C07285=1085.973,384.682,401.818,177.153,26.555,154.362
C07286=1085.978,384.905,401.783,177.157,26.561,154.363
C07287=1085.983,385.128,401.749,177.160,26.567,154.364
C07288=1085.989,385.351,401.714,177.163,26.574,154.365
C07289=1085.995,385.598,401.676,177.166,26.581,154.367
C07290=1086.002,385.844,401.637,177.169,26.588,154.368
C07291=1086.008,386.091,401.600,177.172,26.595,154.369
C07292=1086.014,386.339,401.561,177.176,26.602,154.371
C07293=1086.020,386.585,401.523,177.179,26.608,154.372
C07294=1086.027,386.832,401.485,177.183,26.615,154.373
C07295=1086.032,387.079,401.447,177.186,26.622,154.374
C07296=1086.039,387.326,401.408,177.189,26.629,154.376
C07297=1086.045,387.573,401.370,177.193,26.637,154.377
C07298=1086.052,387.820,401.331,177.196,26.644,154.378
C07299=1086.057,388.066,401.293,177.200,26.651,154.380
C07300=1086.064,388.314,401.254,177.203,26.658,154.381
C07301=1086.069,388.560,401.216,177.206,26.665,154.383
C07302=1086.076,388.807,401.177,177.210,26.672,154.384
C07303=1086.082,389.054,401.140,177.213,26.680,154.385
C07304=1086.089,389.301,401.101,177.217,26.687,154.387
C07305=1086.095,389.548,401.061,177.220,26.694,154.388
C07306=1086.101,389.795,401.024,177.223,26.701,154.389
C07307=1086.108,390.041,400.985,177.227,26.709,154.391
C07308=1086.115,390.288,400.946,177.230,26.715,154.392
C07309=1086.120,390.535,400.908,177.233,26.723,154.393
C07310=1086.127,390.782,400.869,177.237,26.730,154.395
C07311=1086.133,391.028,400.830,177.240,26.737,154.396
C07312=1086.139,391.276,400.792,177.244,26.745,154.398
C07313=1086.145,391.523,400.753,177.247,26.752,154.399
C07314=1086.152,391.769,400.714,177.250,26.759,154.400
C07315=1086.158,392.016,400.675,177.254,26.767,154.402
C07316=1086.164,392.263,400.636,177.257,26.774,154.403
C07317=1086.171,392.509,400.597,177.260,26.781,154.405
C07318=1086.176,392.757,400.559,177.264,26.789,154.406
C07319=1086.183,393.004,400.520,177.267,26.796,154.408
C07320=1086.189,393.251,400.480,177.270,26.804,154.409
C07321=1086.196,393.497,400.442,177.274,26.812,154.411
C07322=1086.202,393.744,400.403,177.277,26.819,154.412
C07323=1086.208,393.991,400.364,177.280,26.826,154.413
C07324=1086.214,394.237,400.325,177.284,26.834,154.415
C07325=1086.221,394.484,400.286,177.287,26.842,154.416
C07326=1086.227,394.731,400.246,177.290,26.849,154.418
C07327=1086.234,394.978,400.208,177.294,26.857,154.419
C07328=1086.240,395.225,400.168,177.298,26.865,154.421
C07329=1086.246,395.471,400.129,177.301,26.873,154.422
C07330=1086.252,395.718,400.090,177.305,26.880,154.424
C07331=1086.258,395.965,400.050,177.308,26.888,154.425
C07332=1086.265,396.212,400.011,177.311,26.895,154.427
C07333=1086.271,396.459,399.972,177.315,26.903,154.428
C07334=1086.277,396.705,399.933,177.318,26.911,154.430
C07335=1086.284,396.951,399.893,177.321,26.919,154.431
C07336=1086.290,397.199,399.854,177.325,26.927,154.433
C07337=1086.296,397.429,399.817,177.328,26.934,154.434
C07338=1086.302,397.658,399.780,177.331,26.941,154.436
C07339=1086.307,397.887,399.744,177.335,26.949,154.437
C07340=1086.314,398.117,399.707,177.337,26.956,154.439
C07341=1086.319,398.347,399.670,177.340,26.964,154.440
C07342=1086.325,398.577,399.633,177.344,26.971,154.442
C07343=1086.331,398.806,399.597,177.347,26.978,154.443
C07344=1086.337,399.036,399.560,177.351,26.986,154.444
C07345=1086.343,399.283,399.520,177.354,26.994,154.446
C07346=1086.350,399.530,399.480,177.357,27.002,154.448
C07347=1086.356,399.777,399.441,177.360,27.010,154.449
C07348=1086.362,400.023,399.401,177.364,27.018,154.451
C07349=1086.368,400.270,399.361,177.367,27.026,154.453
C07350=1086.375,400.517,399.322,177.371,27.034,154.454
C07351=1086.381,400.764,399.282,177.374,27.043,154.456
C07352=1086.388,401.010,399.242,177.378,27.050,154.457
C07353=1086.394,401.257,399.202,177.381,27.059,154.459
C07354=1086.400,401.504,399.162,177.384,27.067,154.461
C07355=1086.407,401.750,399.122,177.388,27.075,154.462
C07356=1086.413,401.997,399.082,177.392,27.084,154.464
C07357=1086.419,402.244,399.043,177.395,27.092,154.466
C07358=1086.425,402.491,399.003,177.398,27.100,154.467
C07359=1086.432,402.737,398.962,177.402,27.108,154.469
C07360=1086.438,402.984,398.922,177.406,27.117,154.471
C07361=1086.445,403.230,398.882,177.409,27.125,154.472
C07362=1086.451,403.477,398.843,177.412,27.133,154.474
C07363=1086.457,403.724,398.803,177.416,27.142,154.476
C07364=1086.463,403.970,398.762,177.420,27.150,154.477
C07365=1086.470,404.217,398.722,177.423,27.159,154.479
C07366=1086.477,404.464,398.682,177.427,27.168,154.481
C07367=1086.483,404.711,398.642,177.430,27.176,154.482
C07368=1086.490,404.957,398.601,177.433,27.184,154.484
C07369=1086.496,405.204,398.561,177.437,27.193,154.486
C07370=1086.502,405.450,398.521,177.441,27.202,154.488
C07371=1086.509,405.697,398.481,177.444,27.211,154.489
C07372=1086.515,405.944,398.440,177.447,27.219,154.491
C07373=1086.521,406.191,398.400,177.451,27.228,154.493
C07374=1086.528,406.437,398.360,177.455,27.236,154.495
C07375=1086.534,406.684,398.319,177.459,27.245,154.496
C07376=1086.540,406.930,398.279,177.462,27.254,154.498
C07377=1086.547,407.177,398.237,177.465,27.263,154.500
C07378=1086.553,407.424,398.197,177.469,27.272,154.502
C07379=1086.560,407.670,398.157,177.472,27.281,154.504
C07380=1086.566,407.917,398.117,177.476,27.290,154.505
C07381=1086.573,408.164,398.075,177.480,27.299,154.507
C07382=1086.579,408.410,398.035,177.483,27.307,154.509
C07383=1086.585,408.657,397.994,177.487,27.316,154.511
C07384=1086.591,408.903,397.953,177.490,27.325,154.513
C07385=1086.598,409.150,397.913,177.494,27.335,154.515
C07386=1086.604,409.397,397.872,177.497,27.343,154.516
C07387=1086.611,409.643,397.831,177.501,27.352,154.518
C07388=1086.616,409.890,397.791,177.505,27.362,154.520
C07389=1086.624,410.136,397.749,177.508,27.371,154.522
C07390=1086.630,410.383,397.709,177.512,27.380,154.524
C07391=1086.636,410.629,397.668,177.515,27.389,154.526
C07392=1086.643,410.876,397.627,177.519,27.398,154.528
C07393=1086.649,411.106,397.589,177.523,27.407,154.529
C07394=1086.655,411.336,397.550,177.526,27.415,154.531
C07395=1086.661,411.567,397.512,177.529,27.424,154.533
C07396=1086.667,411.797,397.474,177.532,27.433,154.535
C07397=1086.673,412.028,397.435,177.536,27.442,154.537
C07398=1086.679,412.258,397.396,177.540,27.451,154.538
C07399=1086.685,412.489,397.359,177.543,27.459,154.540
C07400=1086.691,412.719,397.320,177.546,27.468,154.542
C07401=1086.698,412.966,397.279,177.550,27.478,154.544
C07402=1086.704,413.212,397.238,177.553,27.487,154.546
C07403=1086.712,413.458,397.196,177.558,27.496,154.548
C07404=1086.717,413.705,397.155,177.561,27.505,154.550
C07405=1086.724,413.952,397.114,177.565,27.515,154.552
C07406=1086.730,414.198,397.073,177.568,27.525,154.554
C07407=1086.738,414.445,397.032,177.572,27.534,154.556
C07408=1086.744,414.691,396.990,177.576,27.544,154.558
C07409=1086.751,414.937,396.949,177.579,27.553,154.560
C07410=1086.757,415.184,396.908,177.583,27.563,154.562
C07411=1086.763,415.431,396.866,177.587,27.573,154.564
C07412=1086.770,415.676,396.825,177.590,27.582,154.566
C07413=1086.777,415.923,396.783,177.595,27.592,154.568
C07414=1086.784,416.170,396.742,177.599,27.602,154.570
C07415=1086.790,416.416,396.700,177.602,27.612,154.572
C07416=1086.797,416.662,396.658,177.606,27.622,154.574
C07417=1086.803,416.909,396.616,177.610,27.632,154.576
C07418=1086.809,417.156,396.574,177.613,27.641,154.578
C07419=1086.816,417.401,396.534,177.617,27.652,154.580
C07420=1086.823,417.648,396.491,177.621,27.662,154.582
C07421=1086.829,417.895,396.449,177.624,27.671,154.584
C07422=1086.835,418.141,396.408,177.628,27.682,154.587
C07423=1086.842,418.388,396.366,177.632,27.692,154.589
C07424=1086.848,418.633,396.324,177.636,27.702,154.591
C07425=1086.855,418.880,396.283,177.639,27.712,154.593
C07426=1086.862,419.126,396.240,177.643,27.722,154.595
C07427=1086.868,419.372,396.199,177.647,27.733,154.597
C07428=1086.875,419.619,396.156,177.651,27.743,154.599
C07429=1086.882,419.866,396.114,177.654,27.753,154.602
C07430=1086.888,420.112,396.072,177.658,27.764,154.604
C07431=1086.894,420.358,396.030,177.662,27.774,154.606
C07432=1086.901,420.604,395.988,177.666,27.784,154.608
C07433=1086.909,420.851,395.946,177.670,27.795,154.610
C07434=1086.915,421.097,395.904,177.673,27.805,154.613
C07435=1086.922,421.343,395.862,177.677,27.815,154.615
C07436=1086.928,421.590,395.820,177.681,27.826,154.617
C07437=1086.935,421.836,395.777,177.685,27.836,154.619
C07438=1086.942,422.082,395.735,177.689,27.847,154.622
C07439=1086.949,422.329,395.692,177.693,27.858,154.624
C07440=1086.955,422.575,395.651,177.697,27.868,154.626
C07441=1086.962,422.821,395.608,177.700,27.879,154.628
C07442=1086.968,423.067,395.566,177.704,27.890,154.631
C07443=1086.975,423.314,395.523,177.708,27.901,154.633
C07444=1086.981,423.560,395.480,177.712,27.912,154.635
C07445=1086.988,423.806,395.438,177.716,27.922,154.638
C07446=1086.995,424.052,395.395,177.720,27.933,154.640
C07447=1087.001,424.298,395.353,177.724,27.944,154.642
C07448=1087.008,424.545,395.310,177.728,27.955,154.645
C07449=1087.015,424.783,395.269,177.732,27.966,154.647
C07450=1087.021,425.021,395.228,177.735,27.976,154.649
C07451=1087.028,425.260,395.186,177.739,27.987,154.651
C07452=1087.034,425.497,395.145,177.743,27.998,154.654
C07453=1087.041,425.736,395.104,177.748,28.009,154.656
C07454=1087.047,425.973,395.062,177.751,28.019,154.658
C07455=1087.054,426.212,395.021,177.755,28.030,154.661
C07456=1087.060,426.451,394.979,177.759,28.041,154.663
C07457=1087.067,426.697,394.936,177.763,28.052,154.665
C07458=1087.074,426.943,394.893,177.767,28.063,154.668
C07459=1087.081,427.189,394.850,177.771,28.074,154.670
C07460=1087.087,427.435,394.807,177.774,28.086,154.673
C07461=1087.094,427.681,394.764,177.778,28.097,154.675
C07462=1087.101,427.927,394.721,177.782,28.108,154.678
C07463=1087.108,428.173,394.678,177.786,28.120,154.680
C07464=1087.114,428.420,394.635,177.790,28.131,154.683
C07465=1087.121,428.665,394.592,177.795,28.143,154.685
C07466=1087.128,428.912,394.549,177.799,28.154,154.688
C07467=1087.134,429.158,394.505,177.803,28.166,154.690
C07468=1087.141,429.404,394.463,177.807,28.178,154.693
C07469=1087.148,429.650,394.419,177.811,28.190,154.695
C07470=1087.155,429.896,394.376,177.815,28.201,154.698
C07471=1087.161,430.141,394.332,177.819,28.213,154.700
C07472=1087.168,430.388,394.289,177.823,28.225,154.703
C07473=1087.175,430.634,394.246,177.827,28.236,154.706
C07474=1087.182,430.880,394.202,177.832,28.249,154.708
C07475=1087.189,431.126,394.158,177.836,28.261,154.711
C07476=1087.196,431.372,394.116,177.839,28.273,154.714
C07477=1087.202,431.618,394.072,177.843,28.284,154.716
C07478=1087.209,431.864,394.028,177.847,28.297,154.719
C07479=1087.216,432.110,393.985,177.852,28.309,154.721
C07480=1087.223,432.357,393.940,177.856,28.321,154.724
C07481=1087.230,432.602,393.897,177.860,28.333,154.727
C07482=1087.236,432.848,393.853,177.864,28.345,154.729
C07483=1087.243,433.094,393.810,177.869,28.357,154.732
C07484=1087.250,433.341,393.766,177.873,28.370,154.735
C07485=1087.257,433.586,393.721,177.877,28.382,154.738
C07486=1087.264,433.832,393.677,177.881,28.394,154.740
C07487=1087.271,434.078,393.634,177.885,28.407,154.743
C07488=1087.278,434.324,393.590,177.889,28.420,154.746
C07489=1087.284,434.570,393.546,177.893,28.432,154.749
C07490=1087.291,434.816,393.502,177.897,28.444,154.751
C07491=1087.297,435.062,393.458,177.902,28.457,154.754
C07492=1087.305,435.308,393.414,177.906,28.470,154.757
C07493=1087.312,435.553,393.369,177.910,28.483,154.760
C07494=1087.318,435.799,393.326,177.915,28.495,154.763
C07495=1087.326,436.045,393.281,177.919,28.508,154.765
C07496=1087.332,436.291,393.237,177.922,28.521,154.768
C07497=1087.339,436.537,393.192,177.927,28.534,154.771
C07498=1087.346,436.783,393.149,177.931,28.547,154.774
C07499=1087.353,437.028,393.104,177.936,28.560,154.777
C07500=1087.360,437.275,393.060,177.940,28.573,154.780
C07501=1087.367,437.520,393.015,177.944,28.586,154.783
C07502=1087.374,437.766,392.970,177.949,28.599,154.786
C07503=1087.381,438.012,392.926,177.952,28.612,154.789
C07504=1087.388,438.258,392.882,177.957,28.625,154.792
C07505=1087.395,438.502,392.837,177.961,28.638,154.795
C07506=1087.402,438.746,392.793,177.966,28.652,154.797
C07507=1087.409,438.990,392.749,177.970,28.665,154.800
C07508=1087.416,439.234,392.704,177.974,28.678,154.803
C07509=1087.423,439.478,392.660,177.979,28.691,154.806
C07510=1087.430,439.723,392.616,177.983,28.704,154.809
C07511=1087.438,439.967,392.572,177.988,28.718,154.812
C07512=1087.444,440.211,392.527,177.991,28.731,154.815
C07513=1087.451,440.457,392.482,177.996,28.745,154.818
C07514=1087.458,440.702,392.437,178.000,28.758,154.822
C07515=1087.465,440.948,392.393,178.005,28.772,154.825
C07516=1087.473,441.194,392.348,178.009,28.786,154.828
C07517=1087.479,441.440,392.302,178.014,28.800,154.831
C07518=1087.486,441.685,392.257,178.019,28.814,154.834
C07519=1087.493,441.931,392.212,178.022,28.828,154.837
C07520=1087.500,442.177,392.167,178.027,28.842,154.840
C07521=1087.508,442.422,392.122,178.031,28.855,154.843
C07522=1087.515,442.667,392.077,178.036,28.869,154.847
C07523=1087.521,442.914,392.032,178.041,28.884,154.850
C07524=1087.529,443.159,391.986,178.045,28.898,154.853
C07525=1087.536,443.405,391.941,178.050,28.912,154.856
C07526=1087.543,443.650,391.895,178.054,28.927,154.860
C07527=1087.550,443.896,391.850,178.058,28.941,154.863
C07528=1087.558,444.142,391.805,178.063,28.955,154.866
C07529=1087.564,444.387,391.760,178.068,28.970,154.869
C07530=1087.571,444.633,391.714,178.072,28.984,154.873
C07531=1087.579,444.878,391.668,178.077,28.999,154.876
C07532=1087.586,445.124,391.623,178.081,29.013,154.879
C07533=1087.593,445.370,391.577,178.085,29.028,154.883
C07534=1087.601,445.616,391.531,178.089,29.042,154.886
C07535=1087.607,445.861,391.486,178.092,29.057,154.890
C07536=1087.614,446.107,391.440,178.096,29.071,154.893
C07537=1087.621,446.352,391.394,178.099,29.085,154.896
C07538=1087.629,446.598,391.349,178.102,29.100,154.900
C07539=1087.636,446.844,391.302,178.105,29.114,154.903
C07540=1087.643,447.089,391.257,178.108,29.129,154.907
C07541=1087.650,447.335,391.210,178.111,29.143,154.910
C07542=1087.658,447.580,391.165,178.113,29.158,154.914
C07543=1087.665,447.826,391.119,178.115,29.172,154.917
C07544=1087.673,448.071,391.073,178.117,29.187,154.921
C07545=1087.679,448.317,391.027,178.119,29.201,154.924
C07546=1087.687,448.563,390.981,178.120,29.215,154.928
C07547=1087.694,448.808,390.935,178.122,29.229,154.931
C07548=1087.701,449.054,390.888,178.123,29.244,154.935
C07549=1087.708,449.299,390.843,178.124,29.258,154.938
C07550=1087.716,449.544,390.797,178.125,29.272,154.942
C07551=1087.724,449.789,390.751,178.126,29.286,154.945
C07552=1087.735,450.036,390.706,178.127,29.299,154.948
C07553=1087.357,450.027,390.509,178.088,29.488,155.000
C07554=1087.346,449.781,390.554,178.087,29.475,154.997
C07555=1087.338,449.535,390.600,178.086,29.461,154.993
C07556=1087.330,449.290,390.646,178.085,29.447,154.990
C07557=1087.323,449.046,390.691,178.084,29.433,154.986
C07558=1087.314,448.745,390.748,178.082,29.416,154.982
C07559=1087.305,448.446,390.804,178.080,29.398,154.978
C07560=1087.296,448.146,390.861,178.077,29.380,154.973
C07561=1087.287,447.846,390.917,178.076,29.363,154.969
C07562=1087.280,447.601,390.963,178.073,29.348,154.965
C07563=1087.273,447.355,391.009,178.071,29.334,154.962
C07564=1087.265,447.110,391.055,178.069,29.320,154.958
C07565=1087.258,446.864,391.101,178.066,29.305,154.955
C07566=1087.251,446.618,391.147,178.062,29.291,154.952
C07567=1087.244,446.373,391.193,178.059,29.276,154.948
C07568=1087.236,446.127,391.239,178.055,29.261,154.945
C07569=1087.230,445.882,391.285,178.052,29.247,154.941
C07570=1087.222,445.637,391.330,178.048,29.233,154.938
C07571=1087.215,445.391,391.377,178.045,29.218,154.934
C07572=1087.208,445.145,391.421,178.040,29.203,154.931
C07573=1087.200,444.899,391.467,178.036,29.188,154.928
C07574=1087.194,444.654,391.513,178.032,29.174,154.924
C07575=1087.186,444.408,391.558,178.027,29.160,154.921
C07576=1087.179,444.162,391.604,178.022,29.145,154.918
C07577=1087.172,443.917,391.650,178.018,29.131,154.914
C07578=1087.165,443.671,391.695,178.013,29.117,154.911
C07579=1087.157,443.426,391.740,178.008,29.102,154.908
C07580=1087.150,443.180,391.787,178.004,29.088,154.905
C07581=1087.144,442.935,391.831,177.999,29.074,154.901
C07582=1087.136,442.689,391.876,177.994,29.059,154.898
C07583=1087.129,442.443,391.922,177.990,29.045,154.895
C07584=1087.123,442.197,391.967,177.985,29.031,154.892
C07585=1087.115,441.952,392.013,177.981,29.017,154.889
C07586=1087.108,441.706,392.058,177.976,29.003,154.885
C07587=1087.100,441.460,392.102,177.972,28.990,154.882
C07588=1087.093,441.215,392.148,177.967,28.976,154.879
C07589=1087.086,440.969,392.193,177.962,28.962,154.876
C07590=1087.080,440.724,392.238,177.958,28.948,154.873
C07591=1087.073,440.477,392.283,177.953,28.934,154.870
C07592=1087.065,440.231,392.328,177.949,28.921,154.867
C07593=1087.059,439.986,392.372,177.945,28.907,154.864
C07594=1087.053,439.776,392.411,177.941,28.896,154.861
C07595=1087.046,439.566,392.449,177.937,28.884,154.858
C07596=1087.040,439.356,392.488,177.934,28.873,154.856
C07597=1087.034,439.146,392.525,177.929,28.861,154.853
C07598=1087.028,438.936,392.563,177.926,28.850,154.851
C07599=1087.022,438.725,392.603,177.922,28.839,154.848
C07600=1087.016,438.515,392.640,177.919,28.827,154.846
C07601=1087.010,438.305,392.678,177.914,28.816,154.843
C07602=1087.003,438.059,392.723,177.910,28.803,154.840
C07603=1086.995,437.814,392.767,177.905,28.789,154.837
C07604=1086.988,437.568,392.812,177.902,28.776,154.834
C07605=1086.981,437.322,392.856,177.897,28.763,154.831
C07606=1086.975,437.076,392.901,177.893,28.750,154.828
C07607=1086.967,436.830,392.946,177.889,28.737,154.826
C07608=1086.961,436.584,392.989,177.884,28.724,154.823
C07609=1086.954,436.339,393.034,177.880,28.711,154.820
C07610=1086.947,436.093,393.079,177.876,28.699,154.817
C07611=1086.940,435.847,393.122,177.871,28.685,154.814
C07612=1086.932,435.601,393.167,177.867,28.673,154.811
C07613=1086.926,435.355,393.211,177.863,28.660,154.808
C07614=1086.920,435.109,393.255,177.858,28.647,154.806
C07615=1086.912,434.863,393.300,177.854,28.635,154.803
C07616=1086.905,434.618,393.343,177.850,28.622,154.800
C07617=1086.898,434.372,393.388,177.845,28.609,154.797
C07618=1086.891,434.126,393.432,177.841,28.597,154.794
C07619=1086.885,433.880,393.476,177.837,28.585,154.792
C07620=1086.878,433.634,393.519,177.833,28.572,154.789
C07621=1086.871,433.389,393.563,177.828,28.560,154.786
C07622=1086.864,433.142,393.608,177.824,28.547,154.783
C07623=1086.858,432.896,393.651,177.820,28.535,154.781
C07624=1086.851,432.650,393.695,177.816,28.523,154.778
C07625=1086.843,432.404,393.739,177.811,28.510,154.775
C07626=1086.837,432.158,393.783,177.807,28.498,154.773
C07627=1086.830,431.912,393.826,177.803,28.486,154.770
C07628=1086.823,431.666,393.870,177.799,28.474,154.767
C07629=1086.816,431.420,393.913,177.795,28.462,154.765
C07630=1086.809,431.174,393.957,177.790,28.450,154.762
C07631=1086.802,430.928,394.001,177.786,28.438,154.760
C07632=1086.796,430.682,394.044,177.782,28.426,154.757
C07633=1086.788,430.436,394.088,177.778,28.414,154.754
C07634=1086.782,430.190,394.131,177.774,28.403,154.752
C07635=1086.775,429.944,394.174,177.770,28.391,154.749
C07636=1086.768,429.697,394.218,177.766,28.379,154.746
C07637=1086.761,429.452,394.262,177.761,28.367,154.744
C07638=1086.755,429.205,394.305,177.757,28.355,154.741
C07639=1086.748,428.959,394.348,177.753,28.343,154.739
C07640=1086.741,428.713,394.392,177.749,28.332,154.736
C07641=1086.734,428.467,394.434,177.745,28.321,154.734
C07642=1086.728,428.221,394.478,177.741,28.309,154.731
C07643=1086.721,427.975,394.521,177.737,28.298,154.729
C07644=1086.714,427.729,394.564,177.733,28.286,154.726
C07645=1086.707,427.483,394.607,177.729,28.275,154.724
C07646=1086.701,427.237,394.650,177.725,28.263,154.721
C07647=1086.694,426.991,394.693,177.721,28.252,154.719
C07648=1086.687,426.745,394.736,177.717,28.241,154.717
C07649=1086.680,426.499,394.779,177.713,28.230,154.714
C07650=1086.673,426.259,394.821,177.709,28.218,154.712
C07651=1086.666,426.021,394.863,177.705,28.208,154.709
C07652=1086.660,425.782,394.904,177.700,28.197,154.707
C07653=1086.654,425.543,394.946,177.697,28.186,154.705
C07654=1086.647,425.305,394.987,177.693,28.175,154.702
C07655=1086.641,425.065,395.028,177.689,28.165,154.700
C07656=1086.634,424.827,395.069,177.685,28.154,154.698
C07657=1086.628,424.588,395.112,177.682,28.143,154.695
C07658=1086.621,424.342,395.154,177.678,28.133,154.693
C07659=1086.614,424.095,395.197,177.674,28.121,154.691
C07660=1086.607,423.849,395.239,177.670,28.110,154.688
C07661=1086.601,423.603,395.282,177.666,28.100,154.686
C07662=1086.594,423.357,395.324,177.662,28.089,154.684
C07663=1086.588,423.111,395.367,177.658,28.078,154.682
C07664=1086.581,422.864,395.410,177.654,28.067,154.679
C07665=1086.575,422.618,395.452,177.649,28.056,154.677
C07666=1086.568,422.372,395.495,177.646,28.046,154.675
C07667=1086.561,422.126,395.537,177.642,28.035,154.672
C07668=1086.555,421.880,395.579,177.638,28.025,154.670
C07669=1086.548,421.633,395.621,177.634,28.014,154.668
C07670=1086.541,421.387,395.664,177.630,28.003,154.666
C07671=1086.534,421.141,395.706,177.626,27.993,154.663
C07672=1086.527,420.894,395.749,177.623,27.983,154.661
C07673=1086.521,420.647,395.791,177.619,27.972,154.659
C07674=1086.515,420.402,395.833,177.615,27.962,154.657
C07675=1086.508,420.155,395.875,177.611,27.951,154.654
C07676=1086.500,419.909,395.917,177.607,27.941,154.652
C07677=1086.494,419.663,395.959,177.603,27.931,154.650
C07678=1086.488,419.416,396.001,177.599,27.920,154.648
C07679=1086.481,419.170,396.043,177.595,27.910,154.646
C07680=1086.474,418.923,396.085,177.591,27.900,154.644
C07681=1086.468,418.678,396.127,177.588,27.890,154.641
C07682=1086.461,418.431,396.169,177.584,27.879,154.639
C07683=1086.454,418.185,396.211,177.580,27.869,154.637
C07684=1086.448,417.939,396.252,177.576,27.859,154.635
C07685=1086.441,417.692,396.294,177.573,27.849,154.633
C07686=1086.435,417.445,396.337,177.569,27.839,154.631
C07687=1086.429,417.199,396.378,177.564,27.829,154.629
C07688=1086.422,416.952,396.420,177.561,27.819,154.627
C07689=1086.415,416.706,396.461,177.557,27.809,154.625
C07690=1086.408,416.460,396.503,177.553,27.799,154.622
C07691=1086.402,416.213,396.545,177.550,27.789,154.620
C07692=1086.396,415.967,396.587,177.546,27.780,154.618
C07693=1086.389,415.720,396.628,177.542,27.770,154.616
C07694=1086.383,415.474,396.669,177.538,27.760,154.614
C07695=1086.376,415.227,396.711,177.534,27.750,154.612
C07696=1086.369,414.981,396.752,177.531,27.741,154.610
C07697=1086.363,414.734,396.794,177.527,27.731,154.608
C07698=1086.356,414.488,396.835,177.523,27.721,154.606
C07699=1086.350,414.242,396.876,177.520,27.712,154.604
C07700=1086.342,413.995,396.918,177.516,27.702,154.602
C07701=1086.336,413.749,396.959,177.512,27.693,154.600
C07702=1086.329,413.502,397.000,177.508,27.683,154.598
C07703=1086.323,413.256,397.042,177.504,27.673,154.596
C07704=1086.316,413.009,397.083,177.501,27.664,154.594
C07705=1086.310,412.763,397.125,177.497,27.654,154.592
C07706=1086.303,412.531,397.163,177.493,27.646,154.591
C07707=1086.297,412.301,397.201,177.490,27.637,154.589
C07708=1086.292,412.070,397.240,177.487,27.628,154.587
C07709=1086.285,411.839,397.279,177.483,27.620,154.585
C07710=1086.279,411.608,397.316,177.479,27.611,154.583
C07711=1086.273,411.377,397.356,177.476,27.602,154.582
C07712=1086.267,411.146,397.394,177.473,27.593,154.580
C07713=1086.260,410.915,397.433,177.469,27.584,154.578
C07714=1086.255,410.668,397.473,177.466,27.575,154.576
C07715=1086.248,410.423,397.514,177.462,27.566,154.574
C07716=1086.242,410.175,397.555,177.459,27.557,154.572
C07717=1086.235,409.929,397.596,177.455,27.548,154.570
C07718=1086.229,409.683,397.636,177.451,27.539,154.568
C07719=1086.222,409.436,397.678,177.447,27.530,154.567
C07720=1086.216,409.189,397.718,177.444,27.520,154.565
C07721=1086.210,408.943,397.760,177.440,27.511,154.563
C07722=1086.203,408.696,397.800,177.437,27.502,154.561
C07723=1086.196,408.450,397.841,177.433,27.493,154.559
C07724=1086.191,408.203,397.882,177.429,27.484,154.557
C07725=1086.184,407.956,397.922,177.426,27.476,154.556
C07726=1086.178,407.710,397.964,177.423,27.466,154.554
C07727=1086.171,407.463,398.004,177.419,27.457,154.552
C07728=1086.165,407.217,398.044,177.415,27.449,154.550
C07729=1086.158,406.970,398.084,177.411,27.440,154.548
C07730=1086.152,406.723,398.126,177.408,27.431,154.547
C07731=1086.146,406.477,398.166,177.405,27.422,154.545
C07732=1086.139,406.230,398.206,177.400,27.413,154.543
C07733=1086.133,405.984,398.246,177.397,27.405,154.541
C07734=1086.126,405.737,398.287,177.394,27.396,154.539
C07735=1086.120,405.490,398.328,177.390,27.387,154.538
C07736=1086.114,405.243,398.368,177.386,27.379,154.536
C07737=1086.107,404.997,398.408,177.383,27.370,154.534
C07738=1086.101,404.750,398.448,177.379,27.362,154.533
C07739=1086.095,404.503,398.488,177.376,27.353,154.531
C07740=1086.088,404.256,398.529,177.372,27.345,154.529
C07741=1086.081,404.010,398.569,177.369,27.336,154.527
C07742=1086.075,403.763,398.609,177.365,27.327,154.526
C07743=1086.069,403.517,398.649,177.362,27.319,154.524
C07744=1086.062,403.270,398.689,177.358,27.311,154.522
C07745=1086.056,403.024,398.730,177.355,27.302,154.520
C07746=1086.049,402.777,398.770,177.351,27.294,154.519
C07747=1086.043,402.530,398.809,177.347,27.285,154.517
C07748=1086.036,402.283,398.850,177.344,27.277,154.515
C07749=1086.030,402.036,398.890,177.341,27.269,154.514
C07750=1086.024,401.790,398.930,177.337,27.261,154.512
C07751=1086.017,401.543,398.970,177.333,27.252,154.511
C07752=1086.011,401.296,399.010,177.330,27.244,154.509
C07753=1086.005,401.050,399.050,177.327,27.236,154.507
C07754=1085.998,400.803,399.090,177.323,27.228,154.506
C07755=1085.992,400.556,399.129,177.319,27.219,154.504
C07756=1085.985,400.310,399.169,177.316,27.211,154.502
C07757=1085.979,400.063,399.208,177.313,27.203,154.501
C07758=1085.973,399.816,399.248,177.309,27.195,154.499
C07759=1085.967,399.569,399.288,177.306,27.187,154.497
C07760=1085.960,399.322,399.328,177.303,27.179,154.496
C07761=1085.954,399.075,399.367,177.298,27.170,154.494
C07762=1085.948,398.845,399.404,177.296,27.163,154.493
C07763=1085.942,398.615,399.441,177.292,27.156,154.491
C07764=1085.936,398.385,399.479,177.289,27.148,154.490
C07765=1085.931,398.156,399.515,177.286,27.141,154.488
C07766=1085.925,397.925,399.552,177.283,27.134,154.487
C07767=1085.918,397.695,399.589,177.280,27.126,154.486
C07768=1085.913,397.465,399.626,177.276,27.119,154.484
C07769=1085.907,397.235,399.663,177.273,27.111,154.483
C07770=1085.900,396.988,399.702,177.269,27.103,154.481
C07771=1085.894,396.741,399.741,177.266,27.096,154.480
C07772=1085.888,396.493,399.781,177.263,27.088,154.478
C07773=1085.882,396.248,399.821,177.259,27.080,154.476
C07774=1085.875,396.001,399.859,177.256,27.072,154.475
C07775=1085.869,395.754,399.899,177.253,27.065,154.473
C07776=1085.863,395.507,399.938,177.249,27.057,154.472
C07777=1085.856,395.260,399.977,177.246,27.049,154.470
C07778=1085.850,395.014,400.017,177.242,27.041,154.469
C07779=1085.844,394.767,400.056,177.238,27.033,154.467
C07780=1085.838,394.520,400.095,177.235,27.026,154.466
C07781=1085.831,394.273,400.134,177.232,27.018,154.464
C07782=1085.825,394.026,400.173,177.228,27.011,154.463
C07783=1085.818,393.780,400.212,177.225,27.003,154.462
C07784=1085.812,393.533,400.251,177.221,26.995,154.460
C07785=1085.806,393.286,400.290,177.218,26.988,154.459
C07786=1085.800,393.039,400.330,177.215,26.980,154.457
C07787=1085.793,392.793,400.368,177.211,26.973,154.456
C07788=1085.787,392.546,400.407,177.208,26.965,154.454
C07789=1085.780,392.299,400.446,177.204,26.958,154.453
C07790=1085.775,392.052,400.485,177.201,26.950,154.451
C07791=1085.768,391.805,400.523,177.198,26.943,154.450
C07792=1085.762,391.558,400.563,177.194,26.935,154.448
C07793=1085.756,391.312,400.601,177.191,26.928,154.447
C07794=1085.749,391.065,400.640,177.187,26.921,154.446
C07795=1085.743,390.818,400.679,177.184,26.914,154.444
C07796=1085.737,390.570,400.718,177.181,26.906,154.443
C07797=1085.731,390.324,400.756,177.177,26.899,154.441
C07798=1085.724,390.077,400.795,177.174,26.892,154.440
C07799=1085.717,389.830,400.833,177.170,26.884,154.439
C07800=1085.712,389.583,400.872,177.167,26.877,154.437
C07801=1085.705,389.337,400.911,177.163,26.870,154.436
C07802=1085.699,389.090,400.949,177.160,26.863,154.434
C07803=1085.692,388.843,400.988,177.157,26.856,154.433
C07804=1085.687,388.597,401.027,177.153,26.848,154.432
C07805=1085.680,388.349,401.065,177.150,26.841,154.430
C07806=1085.673,388.102,401.104,177.146,26.834,154.429
C07807=1085.668,387.855,401.141,177.143,26.827,154.428
C07808=1085.661,387.609,401.180,177.139,26.820,154.426
C07809=1085.655,387.362,401.218,177.136,26.812,154.425
C07810=1085.649,387.115,401.257,177.134,26.806,154.424
C07811=1085.643,386.868,401.295,177.130,26.799,154.422
C07812=1085.636,386.621,401.334,177.127,26.792,154.421
C07813=1085.630,386.374,401.372,177.123,26.785,154.420
C07814=1085.624,386.127,401.410,177.120,26.777,154.418
C07815=1085.617,385.881,401.448,177.116,26.771,154.417
C07816=1085.612,385.633,401.487,177.113,26.764,154.416
C07817=1085.606,385.386,401.525,177.109,26.757,154.414
C07818=1085.600,385.163,401.560,177.107,26.750,154.413
C07819=1085.594,384.940,401.594,177.103,26.744,154.412
C07820=1085.589,384.716,401.629,177.101,26.738,154.411
C07821=1085.584,384.493,401.663,177.097,26.731,154.410
C07822=1085.577,384.270,401.698,177.094,26.725,154.409
C07823=1085.572,384.047,401.732,177.092,26.719,154.407
C07824=1085.566,383.823,401.766,177.088,26.713,154.406
C07825=1085.561,383.600,401.800,177.085,26.707,154.405
C07826=1085.554,383.353,401.839,177.082,26.700,154.404
C07827=1085.549,383.107,401.877,177.079,26.693,154.403
C07828=1085.542,382.859,401.915,177.075,26.686,154.401
C07829=1085.536,382.612,401.953,177.072,26.679,154.400
C07830=1085.530,382.366,401.991,177.069,26.673,154.399
C07831=1085.524,382.118,402.029,177.066,26.666,154.398
C07832=1085.518,381.872,402.067,177.062,26.659,154.396
C07833=1085.512,381.625,402.104,177.059,26.653,154.395
C07834=1085.505,381.377,402.142,177.055,26.646,154.394
C07835=1085.499,381.131,402.180,177.052,26.639,154.393
C07836=1085.493,380.883,402.218,177.049,26.633,154.391
C07837=1085.486,380.637,402.255,177.046,26.626,154.390
C07838=1085.481,380.389,402.293,177.042,26.619,154.389
C07839=1085.474,380.142,402.331,177.038,26.613,154.388
C07840=1085.468,379.895,402.368,177.035,26.606,154.386
C07841=1085.462,379.648,402.406,177.032,26.600,154.385
C07842=1085.455,379.401,402.444,177.029,26.593,154.384
C07843=1085.449,379.155,402.481,177.025,26.587,154.383
C07844=1085.444,378.907,402.518,177.022,26.580,154.382
C07845=1085.438,378.660,402.556,177.018,26.574,154.381
C07846=1085.431,378.413,402.594,177.016,26.567,154.379
C07847=1085.425,378.167,402.631,177.012,26.561,154.378
C07848=1085.419,377.919,402.669,177.009,26.554,154.377
C07849=1085.413,377.672,402.706,177.005,26.548,154.376
C07850=1085.406,377.425,402.744,177.003,26.542,154.375
C07851=1085.400,377.178,402.781,176.999,26.535,154.374
C07852=1085.394,376.931,402.819,176.996,26.529,154.372
C07853=1085.389,376.684,402.856,176.992,26.522,154.371
C07854=1085.382,376.437,402.893,176.989,26.516,154.370
C07855=1085.376,376.189,402.930,176.986,26.509,154.369
C07856=1085.370,375.943,402.968,176.982,26.503,154.368
C07857=1085.364,375.696,403.004,176.979,26.496,154.367
C07858=1085.358,375.449,403.042,176.976,26.490,154.365
C07859=1085.352,375.201,403.079,176.973,26.484,154.364
C07860=1085.346,374.955,403.117,176.969,26.477,154.363
C07861=1085.340,374.708,403.153,176.966,26.471,154.362
C07862=1085.333,374.460,403.192,176.963,26.465,154.361
C07863=1085.328,374.213,403.229,176.960,26.459,154.360
C07864=1085.322,373.966,403.265,176.956,26.453,154.359
C07865=1085.316,373.719,403.303,176.953,26.446,154.357
C07866=1085.309,373.472,403.339,176.950,26.440,154.356
C07867=1085.304,373.225,403.376,176.946,26.434,154.355
C07868=1085.297,372.978,403.413,176.944,26.428,154.354
C07869=1085.290,372.730,403.450,176.940,26.422,154.353
C07870=1085.285,372.483,403.487,176.937,26.415,154.352
C07871=1085.278,372.236,403.524,176.933,26.409,154.351
C07872=1085.273,371.989,403.561,176.930,26.404,154.350
C07873=1085.266,371.742,403.598,176.927,26.397,154.349
C07874=1085.261,371.532,403.629,176.924,26.392,154.348
C07875=1085.256,371.323,403.660,176.921,26.387,154.347
C07876=1085.251,371.113,403.691,176.918,26.382,154.346
C07877=1085.245,370.905,403.722,176.915,26.377,154.345
C07878=1085.235,370.486,403.785,176.910,26.366,154.343
C07879=1085.224,370.068,403.847,176.905,26.357,154.342
C07880=1085.219,369.820,403.884,176.901,26.351,154.341
C07881=1085.212,369.573,403.920,176.898,26.345,154.340
C07882=1085.207,369.326,403.957,176.895,26.339,154.338
C07883=1085.200,369.079,403.994,176.892,26.333,154.337
C07884=1085.194,368.832,404.030,176.888,26.327,154.336
C07885=1085.189,368.584,404.067,176.885,26.321,154.335
C07886=1085.182,368.337,404.104,176.882,26.315,154.334
C07887=1085.176,368.090,404.140,176.878,26.309,154.333
C07888=1085.170,367.843,404.177,176.876,26.303,154.332
C07889=1085.164,367.595,404.213,176.872,26.297,154.331
C07890=1085.158,367.348,404.249,176.869,26.291,154.330
C07891=1085.152,367.101,404.286,176.866,26.285,154.329
C07892=1085.146,366.854,404.323,176.862,26.279,154.328
C07893=1085.140,366.607,404.359,176.859,26.274,154.327
C07894=1085.134,366.360,404.395,176.856,26.268,154.326
C07895=1085.129,366.112,404.432,176.853,26.262,154.325
C07896=1085.122,365.865,404.468,176.850,26.256,154.324
C07897=1085.116,365.618,404.504,176.846,26.250,154.323
C07898=1085.110,365.371,404.540,176.843,26.244,154.322
C07899=1085.104,365.123,404.577,176.840,26.239,154.321
C07900=1085.098,364.876,404.613,176.837,26.233,154.320
C07901=1085.092,364.629,404.649,176.833,26.227,154.319
C07902=1085.086,364.381,404.686,176.831,26.222,154.318
C07903=1085.080,364.135,404.721,176.827,26.216,154.317
C07904=1085.074,363.887,404.758,176.823,26.210,154.316
C07905=1085.068,363.640,404.793,176.821,26.205,154.315
C07906=1085.061,363.393,404.830,176.817,26.199,154.314
C07907=1085.055,363.145,404.866,176.814,26.193,154.313
C07908=1085.049,362.898,404.902,176.811,26.188,154.312
C07909=1085.043,362.650,404.938,176.808,26.182,154.311
C07910=1085.037,362.404,404.974,176.804,26.177,154.310
C07911=1085.031,362.156,405.010,176.801,26.170,154.309
C07912=1085.025,361.909,405.045,176.798,26.165,154.308
C07913=1085.019,361.662,405.082,176.794,26.160,154.308
C07914=1085.013,361.414,405.117,176.792,26.154,154.307
C07915=1085.007,361.167,405.154,176.788,26.148,154.306
C07916=1085.001,360.920,405.189,176.785,26.143,154.305
C07917=1084.995,360.672,405.225,176.782,26.137,154.304
C07918=1084.989,360.425,405.261,176.779,26.132,154.303
C07919=1084.983,360.177,405.297,176.775,26.126,154.302
C07920=1084.977,359.930,405.333,176.772,26.121,154.301
C07921=1084.971,359.683,405.368,176.769,26.115,154.300
C07922=1084.965,359.435,405.404,176.766,26.110,154.299
C07923=1084.959,359.188,405.440,176.762,26.104,154.298
C07924=1084.953,358.940,405.476,176.760,26.099,154.297
C07925=1084.947,358.693,405.512,176.756,26.093,154.296
C07926=1084.941,358.446,405.547,176.753,26.088,154.295
C07927=1084.935,358.198,405.582,176.750,26.083,154.294
C07928=1084.925,357.795,405.641,176.745,26.074,154.293
C07929=1084.915,357.394,405.699,176.740,26.065,154.292
C07930=1084.905,356.990,405.756,176.734,26.056,154.290
C07931=1084.896,356.587,405.814,176.729,26.047,154.289
C07932=1084.889,356.340,405.850,176.726,26.043,154.288
C07933=1084.884,356.093,405.885,176.723,26.037,154.287
C07934=1084.878,355.845,405.921,176.720,26.032,154.286
C07935=1084.872,355.598,405.956,176.716,26.027,154.285
C07936=1084.865,355.351,405.991,176.713,26.021,154.284
C07937=1084.860,355.103,406.026,176.710,26.016,154.283
C07938=1084.854,354.856,406.062,176.707,26.011,154.283
C07939=1084.848,354.608,406.097,176.703,26.005,154.282
C07940=1084.841,354.361,406.132,176.701,26.000,154.281
C07941=1084.836,354.114,406.168,176.697,25.995,154.280
C07942=1084.830,353.866,406.203,176.694,25.989,154.279
C07943=1084.825,353.618,406.238,176.691,25.984,154.278
C07944=1084.818,353.371,406.273,176.688,25.979,154.277
C07945=1084.812,353.123,406.309,176.685,25.974,154.277
C07946=1084.807,352.876,406.344,176.681,25.968,154.276
C07947=1084.800,352.628,406.379,176.678,25.963,154.275
C07948=1084.795,352.381,406.414,176.675,25.958,154.274
C07949=1084.788,352.134,406.449,176.672,25.953,154.273
C07950=1084.782,351.886,406.484,176.669,25.948,154.272
C07951=1084.776,351.639,406.519,176.665,25.942,154.271
C07952=1084.770,351.391,406.554,176.663,25.938,154.271
C07953=1084.764,351.144,406.589,176.659,25.932,154.270
C07954=1084.758,350.897,406.625,176.656,25.928,154.269
C07955=1084.752,350.649,406.659,176.653,25.922,154.268
C07956=1084.746,350.402,406.694,176.650,25.917,154.267
C07957=1084.740,350.154,406.728,176.647,25.912,154.266
C07958=1084.734,349.907,406.764,176.643,25.907,154.266
C07959=1084.729,349.659,406.798,176.640,25.902,154.265
C07960=1084.723,349.412,406.834,176.637,25.897,154.264
C07961=1084.717,349.164,406.868,176.634,25.892,154.263
C07962=1084.711,348.917,406.904,176.631,25.887,154.262
C07963=1084.705,348.669,406.938,176.627,25.882,154.262
C07964=1084.699,348.421,406.973,176.624,25.877,154.261
C07965=1084.693,348.174,407.008,176.622,25.872,154.260
C07966=1084.686,347.926,407.042,176.618,25.867,154.259
C07967=1084.681,347.679,407.077,176.615,25.862,154.258
C07968=1084.675,347.431,407.112,176.612,25.857,154.258
C07969=1084.669,347.184,407.146,176.609,25.851,154.257
C07970=1084.663,346.936,407.181,176.606,25.847,154.256
C07971=1084.657,346.689,407.216,176.603,25.842,154.255
C07972=1084.652,346.442,407.250,176.599,25.836,154.254
C07973=1084.645,346.194,407.285,176.596,25.832,154.254
C07974=1084.640,345.946,407.319,176.593,25.827,154.253
C07975=1084.634,345.698,407.354,176.590,25.822,154.252
C07976=1084.627,345.451,407.388,176.587,25.817,154.251
C07977=1084.622,345.204,407.423,176.584,25.812,154.251
C07978=1084.616,344.956,407.458,176.580,25.807,154.250
C07979=1084.610,344.709,407.492,176.578,25.802,154.249
C07980=1084.600,344.309,407.547,176.572,25.794,154.248
C07981=1084.590,343.909,407.603,176.567,25.787,154.246
C07982=1084.581,343.508,407.659,176.562,25.779,154.245
C07983=1084.572,343.109,407.714,176.557,25.771,154.244
C07984=1084.565,342.861,407.748,176.554,25.766,154.243
C07985=1084.559,342.614,407.782,176.551,25.761,154.243
C07986=1084.554,342.366,407.816,176.548,25.757,154.242
C07987=1084.547,342.118,407.851,176.545,25.752,154.241
C07988=1084.541,341.871,407.885,176.542,25.747,154.240
C07989=1084.535,341.624,407.919,176.538,25.742,154.240
C07990=1084.530,341.375,407.954,176.536,25.737,154.239
C07991=1084.524,341.128,407.987,176.533,25.733,154.238
C07992=1084.518,340.880,408.021,176.529,25.728,154.237
C07993=1084.512,340.633,408.055,176.526,25.723,154.237
C07994=1084.506,340.385,408.090,176.523,25.719,154.236
C07995=1084.500,340.138,408.124,176.520,25.714,154.235
C07996=1084.494,339.890,408.158,176.517,25.709,154.234
C07997=1084.488,339.642,408.192,176.514,25.704,154.234
C07998=1084.482,339.395,408.226,176.511,25.700,154.233
C07999=1084.476,339.147,408.260,176.507,25.695,154.232
C08000=1084.470,338.900,408.294,176.504,25.690,154.232
C08001=1084.466,338.652,408.328,176.501,25.685,154.231
C08002=1084.459,338.404,408.362,176.499,25.681,154.230
C08003=1084.453,338.157,408.396,176.495,25.676,154.229
C08004=1084.448,337.909,408.429,176.492,25.671,154.229
C08005=1084.441,337.662,408.463,176.489,25.667,154.228
C08006=1084.435,337.413,408.497,176.486,25.662,154.227
C08007=1084.429,337.166,408.531,176.482,25.657,154.227
C08008=1084.423,336.918,408.565,176.479,25.653,154.226
C08009=1084.418,336.671,408.598,176.477,25.649,154.225
C08010=1084.412,336.423,408.632,176.474,25.644,154.224
C08011=1084.406,336.175,408.666,176.471,25.639,154.224
C08012=1084.400,335.927,408.700,176.467,25.634,154.223
C08013=1084.394,335.680,408.733,176.464,25.630,154.222
C08014=1084.388,335.433,408.767,176.461,25.625,154.222
C08015=1084.382,335.185,408.800,176.458,25.621,154.221
C08016=1084.376,334.937,408.834,176.455,25.616,154.220
C08017=1084.370,334.689,408.868,176.452,25.612,154.220
C08018=1084.365,334.441,408.901,176.449,25.607,154.219
C08019=1084.358,334.194,408.935,176.446,25.603,154.218
C08020=1084.352,333.946,408.968,176.443,25.598,154.217
C08021=1084.347,333.699,409.002,176.439,25.593,154.217
C08022=1084.341,333.451,409.035,176.436,25.589,154.216
C08023=1084.335,333.203,409.069,176.434,25.584,154.216
C08024=1084.329,332.956,409.102,176.431,25.580,154.215
C08025=1084.323,332.708,409.135,176.428,25.576,154.214
C08026=1084.318,332.460,409.169,176.425,25.571,154.214
C08027=1084.312,332.212,409.202,176.421,25.567,154.213
C08028=1084.306,331.965,409.236,176.418,25.562,154.212
C08029=1084.299,331.717,409.269,176.415,25.557,154.211
C08030=1084.294,331.469,409.303,176.412,25.553,154.211
C08031=1084.288,331.221,409.335,176.409,25.549,154.210
C08032=1084.278,330.816,409.390,176.404,25.541,154.209
C08033=1084.268,330.410,409.445,176.399,25.534,154.208
C08034=1084.259,330.005,409.499,176.394,25.527,154.207
C08035=1084.249,329.599,409.553,176.389,25.520,154.206
C08036=1084.242,329.351,409.586,176.386,25.516,154.205
C08037=1084.237,329.103,409.619,176.383,25.511,154.205
C08038=1084.230,328.856,409.652,176.380,25.507,154.204
C08039=1084.225,328.608,409.686,176.377,25.503,154.203
C08040=1084.219,328.360,409.718,176.374,25.499,154.203
C08041=1084.212,328.113,409.751,176.371,25.494,154.202
C08042=1084.207,327.865,409.784,176.367,25.490,154.202
C08043=1084.200,327.617,409.817,176.364,25.485,154.201
C08044=1084.195,327.369,409.850,176.362,25.481,154.200
C08045=1084.189,327.122,409.883,176.359,25.477,154.200
C08046=1084.183,326.874,409.916,176.356,25.473,154.199
C08047=1084.177,326.626,409.949,176.353,25.468,154.198
C08048=1084.171,326.378,409.981,176.350,25.464,154.198
C08049=1084.165,326.130,410.015,176.347,25.460,154.197
C08050=1084.159,325.882,410.047,176.343,25.455,154.197
C08051=1084.153,325.634,410.081,176.340,25.451,154.196
C08052=1084.147,325.387,410.113,176.337,25.447,154.195
C08053=1084.141,325.139,410.146,176.334,25.442,154.195
C08054=1084.136,324.891,410.178,176.331,25.438,154.194
C08055=1084.130,324.644,410.211,176.328,25.434,154.194
C08056=1084.124,324.396,410.245,176.326,25.430,154.193
C08057=1084.118,324.148,410.277,176.323,25.426,154.192
C08058=1084.112,323.900,410.309,176.320,25.421,154.192
C08059=1084.106,323.652,410.343,176.317,25.417,154.191
C08060=1084.100,323.405,410.375,176.313,25.413,154.190
C08061=1084.094,323.156,410.407,176.310,25.408,154.190
C08062=1084.089,322.909,410.440,176.307,25.404,154.189
C08063=1084.083,322.662,410.473,176.304,25.400,154.189
C08064=1084.077,322.413,410.505,176.301,25.396,154.188
C08065=1084.071,322.166,410.538,176.298,25.391,154.187
C08066=1084.065,321.917,410.570,176.295,25.387,154.187
C08067=1084.059,321.670,410.603,176.292,25.383,154.186
C08068=1084.054,321.423,410.636,176.290,25.379,154.186
C08069=1084.048,321.174,410.668,176.286,25.375,154.185
C08070=1084.042,320.927,410.701,176.284,25.370,154.184
C08071=1084.036,320.679,410.733,176.281,25.366,154.184
C08072=1084.031,320.431,410.766,176.278,25.362,154.183
C08073=1084.025,320.183,410.798,176.275,25.358,154.183
C08074=1084.019,319.936,410.831,176.272,25.354,154.182
C08075=1084.013,319.687,410.863,176.269,25.350,154.181
C08076=1084.008,319.439,410.895,176.265,25.345,154.181
C08077=1084.002,319.192,410.928,176.262,25.341,154.180
C08078=1083.996,318.944,410.960,176.259,25.337,154.180
C08079=1083.991,318.696,410.993,176.256,25.333,154.179
C08080=1083.985,318.448,411.025,176.253,25.329,154.178
C08081=1083.979,318.200,411.057,176.250,25.324,154.178
C08082=1083.973,317.953,411.089,176.247,25.320,154.177
C08083=1083.967,317.705,411.121,176.245,25.316,154.177
C08084=1083.957,317.293,411.175,176.240,25.309,154.176
C08085=1083.949,316.880,411.229,176.235,25.302,154.175
C08086=1083.939,316.468,411.283,176.230,25.295,154.174
C08087=1083.930,316.055,411.336,176.225,25.288,154.173
C08088=1083.924,315.807,411.368,176.222,25.284,154.172
C08089=1083.918,315.560,411.400,176.219,25.280,154.172
C08090=1083.912,315.312,411.432,176.216,25.276,154.171
C08091=1083.907,315.065,411.464,176.213,25.272,154.170
C08092=1083.901,314.816,411.496,176.210,25.268,154.170
C08093=1083.895,314.568,411.528,176.207,25.264,154.169
C08094=1083.889,314.320,411.560,176.204,25.260,154.169
C08095=1083.883,314.073,411.592,176.201,25.256,154.168
C08096=1083.877,313.824,411.624,176.198,25.252,154.168
C08097=1083.871,313.576,411.655,176.195,25.248,154.167
C08098=1083.865,313.329,411.687,176.192,25.244,154.167
C08099=1083.859,313.081,411.719,176.189,25.240,154.166
C08100=1083.853,312.832,411.751,176.186,25.236,154.166
C08101=1083.847,312.585,411.782,176.183,25.232,154.165
C08102=1083.841,312.337,411.814,176.180,25.228,154.164
C08103=1083.836,312.090,411.846,176.178,25.224,154.164
C08104=1083.830,311.841,411.878,176.175,25.220,154.163
C08105=1083.823,311.593,411.909,176.172,25.216,154.163
C08106=1083.818,311.346,411.941,176.169,25.213,154.162
C08107=1083.812,311.098,411.973,176.166,25.209,154.162
C08108=1083.806,310.850,412.004,176.163,25.205,154.161
C08109=1083.800,310.602,412.036,176.160,25.201,154.161
C08110=1083.794,310.354,412.068,176.157,25.197,154.160
C08111=1083.788,310.107,412.100,176.154,25.193,154.160
C08112=1083.782,309.858,412.130,176.151,25.189,154.159
C08113=1083.777,309.611,412.162,176.148,25.185,154.159
C08114=1083.771,309.362,412.194,176.145,25.181,154.158
C08115=1083.764,309.115,412.225,176.142,25.177,154.158
C08116=1083.758,308.867,412.257,176.139,25.173,154.157
C08117=1083.753,308.619,412.288,176.136,25.169,154.157
C08118=1083.747,308.371,412.320,176.133,25.165,154.156
C08119=1083.741,308.123,412.351,176.130,25.161,154.155
C08120=1083.735,307.875,412.383,176.127,25.157,154.155
C08121=1083.729,307.627,412.413,176.124,25.153,154.154
C08122=1083.723,307.379,412.446,176.121,25.150,154.154
C08123=1083.718,307.132,412.477,176.118,25.146,154.153
C08124=1083.712,306.884,412.508,176.115,25.142,154.153
C08125=1083.706,306.636,412.540,176.112,25.138,154.152
C08126=1083.701,306.388,412.571,176.109,25.134,154.152
C08127=1083.694,306.139,412.602,176.106,25.130,154.151
C08128=1083.689,305.892,412.634,176.103,25.126,154.151
C08129=1083.683,305.644,412.664,176.101,25.123,154.150
C08130=1083.677,305.396,412.696,176.098,25.119,154.150
C08131=1083.672,305.148,412.728,176.095,25.115,154.149
C08132=1083.665,304.900,412.758,176.092,25.111,154.149
C08133=1083.660,304.652,412.790,176.089,25.107,154.148
C08134=1083.654,304.405,412.820,176.086,25.103,154.148
C08135=1083.648,304.156,412.852,176.083,25.099,154.147
C08136=1083.639,303.746,412.903,176.078,25.093,154.146
C08137=1083.630,303.338,412.955,176.074,25.087,154.146
C08138=1083.620,302.929,413.006,176.069,25.080,154.145
C08139=1083.611,302.519,413.057,176.064,25.074,154.144
C08140=1083.605,302.271,413.088,176.061,25.070,154.143
C08141=1083.599,302.023,413.120,176.058,25.066,154.143
C08142=1083.594,301.775,413.151,176.055,25.062,154.142
C08143=1083.588,301.527,413.181,176.052,25.058,154.142
C08144=1083.582,301.280,413.213,176.050,25.055,154.141
C08145=1083.576,301.031,413.243,176.047,25.051,154.141
C08146=1083.571,300.783,413.274,176.044,25.047,154.140
C08147=1083.565,300.535,413.305,176.041,25.043,154.140
C08148=1083.560,300.288,413.336,176.038,25.039,154.139
C08149=1083.554,300.040,413.367,176.035,25.035,154.139
C08150=1083.548,299.791,413.398,176.032,25.031,154.138
C08151=1083.542,299.543,413.428,176.029,25.027,154.138
C08152=1083.537,299.295,413.459,176.026,25.024,154.137
C08153=1083.531,299.048,413.490,176.024,25.020,154.137
C08154=1083.526,298.800,413.521,176.021,25.016,154.136
C08155=1083.520,298.551,413.552,176.018,25.012,154.136
C08156=1083.515,298.303,413.583,176.015,25.008,154.135
C08157=1083.509,298.055,413.613,176.012,25.005,154.135
C08158=1083.503,297.808,413.644,176.009,25.001,154.134
C08159=1083.498,297.559,413.675,176.006,24.997,154.134
C08160=1083.492,297.311,413.705,176.004,24.994,154.133
C08161=1083.485,297.064,413.736,176.001,24.990,154.133
C08162=1083.480,296.816,413.767,175.998,24.986,154.132
C08163=1083.475,296.568,413.798,175.995,24.982,154.132
C08164=1083.469,296.320,413.828,175.992,24.978,154.131
C08165=1083.462,296.071,413.859,175.989,24.975,154.131
C08166=1083.456,295.824,413.889,175.986,24.971,154.130
C08167=1083.451,295.576,413.920,175.984,24.968,154.130
C08168=1083.446,295.327,413.950,175.981,24.964,154.129
C08169=1083.440,295.079,413.980,175.978,24.960,154.129
C08170=1083.434,294.831,414.010,175.975,24.956,154.128
C08171=1083.428,294.583,414.041,175.972,24.953,154.128
C08172=1083.422,294.335,414.072,175.969,24.949,154.128
C08173=1083.416,294.087,414.102,175.966,24.945,154.127
C08174=1083.410,293.839,414.132,175.964,24.942,154.127
C08175=1083.405,293.592,414.163,175.961,24.938,154.126
C08176=1083.400,293.343,414.193,175.958,24.934,154.126
C08177=1083.394,293.095,414.223,175.955,24.931,154.125
C08178=1083.388,292.846,414.254,175.952,24.927,154.125
C08179=1083.382,292.599,414.284,175.949,24.924,154.124
C08180=1083.376,292.351,414.315,175.947,24.920,154.124
C08181=1083.370,292.102,414.344,175.943,24.916,154.123
C08182=1083.365,291.855,414.375,175.940,24.912,154.123
C08183=1083.359,291.607,414.405,175.937,24.909,154.122
C08184=1083.353,291.359,414.435,175.934,24.905,154.122
C08185=1083.347,291.110,414.465,175.932,24.901,154.121
C08186=1083.342,290.863,414.495,175.929,24.897,154.121
C08187=1083.336,290.615,414.526,175.926,24.894,154.121
C08188=1083.327,290.219,414.574,175.922,24.888,154.120
C08189=1083.317,289.824,414.621,175.917,24.882,154.119
C08190=1083.309,289.429,414.669,175.913,24.877,154.118
C08191=1083.299,289.033,414.717,175.908,24.871,154.118
C08192=1083.293,288.785,414.748,175.905,24.867,154.117
C08193=1083.288,288.537,414.777,175.902,24.863,154.117
C08194=1083.282,288.289,414.807,175.899,24.860,154.116
C08195=1083.276,288.041,414.837,175.897,24.856,154.116
C08196=1083.270,287.793,414.867,175.894,24.853,154.115
C08197=1083.264,287.545,414.897,175.891,24.849,154.115
C08198=1083.258,287.297,414.927,175.888,24.845,154.114
C08199=1083.253,287.049,414.957,175.886,24.842,154.114
C08200=1083.246,286.801,414.986,175.883,24.839,154.114
C08201=1083.241,286.553,415.016,175.880,24.835,154.113
C08202=1083.235,286.304,415.046,175.877,24.831,154.113
C08203=1083.229,286.056,415.076,175.874,24.828,154.112
C08204=1083.224,285.808,415.106,175.872,24.825,154.112
C08205=1083.218,285.560,415.135,175.869,24.820,154.111
C08206=1083.212,285.312,415.165,175.866,24.817,154.111
C08207=1083.206,285.063,415.195,175.863,24.813,154.111
C08208=1083.201,284.815,415.224,175.861,24.810,154.110
C08209=1083.195,284.567,415.255,175.857,24.806,154.110
C08210=1083.189,284.319,415.284,175.854,24.803,154.109
C08211=1083.184,284.071,415.313,175.851,24.799,154.109
C08212=1083.178,283.824,415.343,175.849,24.796,154.108
C08213=1083.173,283.575,415.373,175.846,24.792,154.108
C08214=1083.166,283.327,415.402,175.843,24.788,154.107
C08215=1083.161,283.078,415.432,175.840,24.785,154.107
C08216=1083.155,282.830,415.461,175.838,24.782,154.107
C08217=1083.149,282.582,415.491,175.835,24.777,154.106
C08218=1083.143,282.334,415.521,175.832,24.774,154.106
C08219=1083.138,282.086,415.550,175.829,24.770,154.105
C08220=1083.132,281.837,415.580,175.827,24.767,154.105
C08221=1083.127,281.590,415.608,175.824,24.763,154.104
C08222=1083.121,281.341,415.638,175.821,24.760,154.104
C08223=1083.116,281.093,415.668,175.818,24.756,154.103
C08224=1083.109,280.845,415.697,175.816,24.753,154.103
C08225=1083.103,280.597,415.727,175.813,24.749,154.103
C08226=1083.098,280.349,415.757,175.810,24.746,154.102
C08227=1083.092,280.100,415.786,175.807,24.742,154.102
C08228=1083.087,279.853,415.815,175.804,24.739,154.101
C08229=1083.081,279.605,415.844,175.801,24.735,154.101
C08230=1083.075,279.356,415.874,175.798,24.731,154.100
C08231=1083.069,279.108,415.903,175.796,24.728,154.100
C08232=1083.063,278.859,415.932,175.793,24.725,154.100
C08233=1083.057,278.611,415.961,175.790,24.721,154.099
C08234=1083.052,278.362,415.990,175.787,24.718,154.099
C08235=1083.046,278.115,416.019,175.785,24.715,154.098
C08236=1083.041,277.866,416.049,175.782,24.711,154.098
C08237=1083.034,277.618,416.078,175.779,24.707,154.097
C08238=1083.029,277.370,416.107,175.777,24.704,154.097
C08239=1083.023,277.122,416.136,175.774,24.700,154.097
C08240=1083.014,276.736,416.181,175.769,24.695,154.096
C08241=1083.005,276.351,416.226,175.765,24.689,154.095
C08242=1082.997,275.966,416.271,175.761,24.684,154.095
C08243=1082.988,275.581,416.317,175.757,24.679,154.094
C08244=1082.982,275.332,416.346,175.754,24.675,154.094
C08245=1082.976,275.084,416.375,175.751,24.672,154.093
C08246=1082.971,274.835,416.405,175.748,24.668,154.093
C08247=1082.965,274.588,416.433,175.745,24.665,154.092
C08248=1082.959,274.339,416.462,175.742,24.661,154.092
C08249=1082.953,274.090,416.491,175.740,24.658,154.091
C08250=1082.947,273.842,416.520,175.737,24.654,154.091
C08251=1082.942,273.594,416.548,175.734,24.651,154.091
C08252=1082.936,273.346,416.578,175.732,24.647,154.090
C08253=1082.930,273.098,416.607,175.729,24.644,154.090
C08254=1082.925,272.850,416.635,175.726,24.640,154.089
C08255=1082.919,272.601,416.664,175.724,24.637,154.089
C08256=1082.913,272.352,416.693,175.721,24.634,154.089
C08257=1082.907,272.104,416.722,175.718,24.630,154.088
C08258=1082.902,271.856,416.750,175.716,24.627,154.088
C08259=1082.896,271.608,416.779,175.713,24.623,154.087
C08260=1082.890,271.360,416.808,175.710,24.619,154.087
C08261=1082.885,271.112,416.836,175.707,24.616,154.086
C08262=1082.878,270.864,416.865,175.704,24.613,154.086
C08263=1082.873,270.614,416.894,175.701,24.609,154.086
C08264=1082.868,270.367,416.923,175.699,24.606,154.085
C08265=1082.862,270.118,416.951,175.696,24.603,154.085
C08266=1082.856,269.870,416.980,175.693,24.599,154.084
C08267=1082.850,269.622,417.008,175.691,24.596,154.084
C08268=1082.845,269.373,417.037,175.688,24.592,154.084
C08269=1082.839,269.125,417.066,175.686,24.589,154.083
C08270=1082.833,268.877,417.094,175.683,24.586,154.083
C08271=1082.827,268.628,417.123,175.680,24.582,154.082
C08272=1082.822,268.381,417.151,175.678,24.579,154.082
C08273=1082.816,268.132,417.180,175.674,24.575,154.082
C08274=1082.810,267.883,417.208,175.671,24.572,154.081
C08275=1082.804,267.636,417.237,175.669,24.569,154.081
C08276=1082.798,267.387,417.265,175.666,24.565,154.080
C08277=1082.793,267.139,417.293,175.663,24.562,154.080
C08278=1082.787,266.891,417.323,175.661,24.558,154.080
C08279=1082.781,266.642,417.351,175.658,24.555,154.079
C08280=1082.776,266.394,417.379,175.655,24.551,154.079
C08281=1082.770,266.145,417.407,175.653,24.548,154.078
C08282=1082.764,265.898,417.436,175.650,24.545,154.078
C08283=1082.758,265.649,417.464,175.648,24.542,154.078
C08284=1082.753,265.401,417.492,175.645,24.538,154.077
C08285=1082.747,265.152,417.520,175.642,24.534,154.077
C08286=1082.741,264.903,417.549,175.639,24.531,154.076
C08287=1082.736,264.656,417.577,175.636,24.528,154.076
C08288=1082.730,264.407,417.606,175.633,24.524,154.076
C08289=1082.724,264.159,417.634,175.631,24.521,154.075
C08290=1082.718,263.910,417.662,175.628,24.517,154.075
C08291=1082.713,263.662,417.690,175.626,24.514,154.074
C08292=1082.704,263.279,417.734,175.621,24.509,154.074
C08293=1082.695,262.897,417.776,175.618,24.504,154.073
C08294=1082.685,262.514,417.820,175.613,24.499,154.073
C08295=1082.677,262.132,417.863,175.609,24.494,154.072
C08296=1082.671,261.884,417.891,175.606,24.491,154.072
C08297=1082.665,261.636,417.919,175.603,24.487,154.071
C08298=1082.659,261.387,417.947,175.601,24.484,154.071
C08299=1082.653,261.139,417.975,175.598,24.480,154.071
C08300=1082.648,260.890,418.002,175.595,24.477,154.070
C08301=1082.642,260.642,418.030,175.593,24.474,154.070
C08302=1082.636,260.393,418.058,175.590,24.471,154.069
C08303=1082.630,260.145,418.086,175.588,24.468,154.069
C08304=1082.624,259.896,418.114,175.585,24.464,154.069
C08305=1082.618,259.649,418.142,175.582,24.460,154.068
C08306=1082.612,259.400,418.170,175.580,24.457,154.068
C08307=1082.607,259.152,418.198,175.577,24.454,154.067
C08308=1082.601,258.903,418.226,175.574,24.451,154.067
C08309=1082.595,258.655,418.253,175.571,24.447,154.067
C08310=1082.589,258.406,418.281,175.569,24.444,154.066
C08311=1082.584,258.158,418.309,175.566,24.441,154.066
C08312=1082.577,257.910,418.337,175.563,24.437,154.066
C08313=1082.572,257.661,418.364,175.561,24.434,154.065
C08314=1082.567,257.413,418.392,175.558,24.430,154.065
C08315=1082.560,257.164,418.420,175.556,24.428,154.065
C08316=1082.555,256.916,418.448,175.553,24.424,154.064
C08317=1082.549,256.667,418.476,175.550,24.421,154.064
C08318=1082.543,256.419,418.503,175.547,24.418,154.063
C08319=1082.538,256.171,418.531,175.544,24.414,154.063
C08320=1082.532,255.922,418.559,175.542,24.411,154.063
C08321=1082.526,255.674,418.586,175.539,24.407,154.062
C08322=1082.520,255.425,418.614,175.537,24.404,154.062
C08323=1082.515,255.177,418.641,175.534,24.401,154.061
C08324=1082.509,254.929,418.669,175.532,24.398,154.061
C08325=1082.503,254.680,418.696,175.529,24.394,154.061
C08326=1082.497,254.432,418.724,175.527,24.391,154.060
C08327=1082.492,254.184,418.752,175.524,24.388,154.060
C08328=1082.486,253.934,418.779,175.521,24.384,154.059
C08329=1082.480,253.687,418.807,175.519,24.381,154.059
C08330=1082.475,253.438,418.834,175.515,24.377,154.059
C08331=1082.469,253.190,418.861,175.513,24.374,154.058
C08332=1082.464,252.941,418.889,175.510,24.371,154.058
C08333=1082.458,252.693,418.917,175.508,24.368,154.058
C08334=1082.452,252.444,418.944,175.505,24.364,154.057
C08335=1082.447,252.196,418.972,175.503,24.361,154.057
C08336=1082.441,251.947,418.999,175.500,24.357,154.056
C08337=1082.435,251.699,419.026,175.498,24.354,154.056
C08338=1082.430,251.451,419.054,175.495,24.351,154.056
C08339=1082.424,251.202,419.081,175.493,24.348,154.055
C08340=1082.419,250.953,419.109,175.490,24.344,154.055
C08341=1082.413,250.705,419.135,175.488,24.341,154.054
C08342=1082.408,250.456,419.163,175.484,24.338,154.054
C08343=1082.402,250.209,419.190,175.481,24.334,154.054
C08344=1082.394,249.823,419.232,175.478,24.329,154.053
C08345=1082.385,249.438,419.274,175.474,24.324,154.052
C08346=1082.376,249.052,419.316,175.470,24.318,154.052
C08347=1082.367,248.667,419.359,175.466,24.313,154.051
C08348=1082.361,248.419,419.386,175.463,24.310,154.051
C08349=1082.356,248.170,419.414,175.461,24.307,154.050
C08350=1082.350,247.921,419.441,175.458,24.303,154.050
C08351=1082.345,247.673,419.468,175.456,24.300,154.050
C08352=1082.339,247.424,419.494,175.453,24.297,154.049
C08353=1082.334,247.176,419.522,175.451,24.294,154.049
C08354=1082.328,246.928,419.549,175.448,24.290,154.048
C08355=1082.322,246.680,419.576,175.445,24.287,154.048
C08356=1082.317,246.430,419.603,175.442,24.283,154.048
C08357=1082.311,246.182,419.630,175.440,24.280,154.047
C08358=1082.305,245.933,419.657,175.437,24.277,154.047
C08359=1082.300,245.685,419.684,175.435,24.274,154.047
C08360=1082.294,245.437,419.711,175.432,24.270,154.046
C08361=1082.288,245.189,419.738,175.430,24.267,154.046
C08362=1082.283,244.940,419.765,175.427,24.263,154.045
C08363=1082.277,244.691,419.792,175.425,24.260,154.045
C08364=1082.271,244.443,419.819,175.422,24.257,154.045
C08365=1082.266,244.194,419.846,175.420,24.254,154.044
C08366=1082.260,243.946,419.873,175.417,24.250,154.044
C08367=1082.254,243.697,419.899,175.414,24.247,154.044
C08368=1082.249,243.449,419.926,175.411,24.244,154.043
C08369=1082.244,243.200,419.953,175.409,24.240,154.043
C08370=1082.238,242.952,419.980,175.406,24.237,154.042
C08371=1082.232,242.703,420.007,175.404,24.234,154.042
C08372=1082.226,242.454,420.034,175.401,24.231,154.042
C08373=1082.220,242.206,420.060,175.399,24.227,154.041
C08374=1082.214,241.958,420.087,175.397,24.224,154.041
C08375=1082.209,241.709,420.113,175.394,24.221,154.041
C08376=1082.203,241.460,420.139,175.392,24.218,154.040
C08377=1082.198,241.212,420.167,175.389,24.214,154.040
C08378=1082.192,240.963,420.193,175.386,24.211,154.039
C08379=1082.186,240.715,420.220,175.383,24.208,154.039
C08380=1082.181,240.467,420.247,175.381,24.205,154.039
C08381=1082.175,240.218,420.273,175.378,24.201,154.038
C08382=1082.169,239.969,420.299,175.376,24.198,154.038
C08383=1082.163,239.721,420.326,175.373,24.195,154.038
C08384=1082.158,239.473,420.353,175.371,24.192,154.037
C08385=1082.151,239.223,420.380,175.368,24.188,154.037
C08386=1082.146,238.975,420.405,175.366,24.185,154.036
C08387=1082.140,238.726,420.432,175.364,24.182,154.036
C08388=1082.134,238.478,420.459,175.360,24.179,154.036
C08389=1082.129,238.229,420.485,175.358,24.176,154.035
C08390=1082.123,237.980,420.511,175.355,24.172,154.035
C08391=1082.117,237.732,420.538,175.353,24.169,154.035
C08392=1082.112,237.484,420.565,175.350,24.166,154.034
C08393=1082.106,237.235,420.591,175.348,24.163,154.034
C08394=1082.100,236.986,420.617,175.346,24.159,154.033
C08395=1082.095,236.738,420.644,175.343,24.156,154.033
C08396=1082.086,236.346,420.685,175.339,24.151,154.032
C08397=1082.077,235.953,420.726,175.335,24.145,154.032
C08398=1082.068,235.561,420.768,175.331,24.140,154.031
C08399=1082.059,235.170,420.809,175.327,24.135,154.031
C08400=1082.053,234.921,420.836,175.325,24.132,154.030
C08401=1082.048,234.673,420.861,175.322,24.129,154.030
C08402=1082.042,234.424,420.888,175.319,24.125,154.030
C08403=1082.036,234.175,420.914,175.317,24.122,154.029
C08404=1082.031,233.927,420.941,175.314,24.119,154.029
C08405=1082.025,233.678,420.967,175.312,24.116,154.029
C08406=1082.019,233.429,420.993,175.310,24.113,154.028
C08407=1082.014,233.180,421.019,175.307,24.109,154.028
C08408=1082.008,232.933,421.044,175.305,24.106,154.027
C08409=1082.003,232.684,421.071,175.302,24.103,154.027
C08410=1081.997,232.435,421.097,175.300,24.100,154.027
C08411=1081.991,232.187,421.123,175.298,24.096,154.026
C08412=1081.986,231.938,421.149,175.295,24.093,154.026
C08413=1081.980,231.689,421.175,175.293,24.090,154.025
C08414=1081.974,231.441,421.201,175.289,24.087,154.025
C08415=1081.968,231.192,421.227,175.287,24.083,154.025
C08416=1081.963,230.944,421.254,175.285,24.080,154.024
C08417=1081.958,230.695,421.279,175.282,24.077,154.024
C08418=1081.952,230.447,421.305,175.280,24.074,154.024
C08419=1081.946,230.198,421.331,175.277,24.070,154.023
C08420=1081.940,229.939,421.357,175.275,24.067,154.023
C08421=1081.934,229.680,421.385,175.272,24.063,154.023
C08422=1081.929,229.422,421.412,175.270,24.060,154.022
C08423=1081.922,229.164,421.439,175.267,24.057,154.022
C08424=1081.917,228.915,421.465,175.265,24.054,154.021
C08425=1081.910,228.666,421.490,175.262,24.050,154.021
C08426=1081.906,228.418,421.516,175.259,24.047,154.021
C08427=1081.899,228.170,421.542,175.257,24.044,154.020
C08428=1081.894,227.921,421.568,175.254,24.041,154.020
C08429=1081.888,227.672,421.594,175.252,24.038,154.020
C08430=1081.882,227.423,421.619,175.250,24.034,154.019
C08431=1081.877,227.175,421.645,175.247,24.031,154.019
C08432=1081.871,226.926,421.670,175.245,24.028,154.019
C08433=1081.865,226.677,421.696,175.243,24.025,154.018
C08434=1081.859,226.429,421.722,175.240,24.021,154.018
C08435=1081.853,226.180,421.748,175.238,24.019,154.017
C08436=1081.848,225.932,421.773,175.235,24.015,154.017
C08437=1081.842,225.683,421.799,175.232,24.012,154.017
C08438=1081.837,225.434,421.825,175.230,24.009,154.016
C08439=1081.831,225.185,421.850,175.227,24.005,154.016
C08440=1081.826,224.937,421.876,175.225,24.002,154.016
C08441=1081.820,224.688,421.901,175.223,23.999,154.015
C08442=1081.814,224.439,421.927,175.220,23.995,154.015
C08443=1081.808,224.191,421.952,175.218,23.993,154.015
C08444=1081.803,223.943,421.978,175.216,23.989,154.014
C08445=1081.797,223.694,422.003,175.213,23.986,154.014
C08446=1081.791,223.445,422.029,175.211,23.983,154.013
C08447=1081.786,223.197,422.054,175.209,23.980,154.013
C08448=1081.777,222.806,422.094,175.204,23.974,154.012
C08449=1081.769,222.415,422.134,175.200,23.969,154.012
C08450=1081.760,222.025,422.174,175.197,23.964,154.011
C08451=1081.751,221.634,422.214,175.193,23.959,154.011
C08452=1081.745,221.385,422.239,175.190,23.956,154.010
C08453=1081.739,221.136,422.264,175.188,23.953,154.010
C08454=1081.733,220.887,422.290,175.186,23.950,154.010
C08455=1081.728,220.639,422.315,175.183,23.946,154.009
C08456=1081.721,220.391,422.341,175.181,23.943,154.009
C08457=1081.716,220.141,422.366,175.179,23.940,154.009
C08458=1081.711,219.893,422.391,175.176,23.937,154.008
C08459=1081.704,219.644,422.416,175.174,23.933,154.008
C08460=1081.698,219.396,422.442,175.172,23.931,154.007
C08461=1081.694,219.147,422.466,175.169,23.927,154.007
C08462=1081.687,218.898,422.492,175.166,23.924,154.007
C08463=1081.681,218.650,422.517,175.164,23.921,154.006
C08464=1081.677,218.401,422.542,175.161,23.918,154.006
C08465=1081.670,218.152,422.567,175.159,23.914,154.006
C08466=1081.665,217.904,422.592,175.157,23.911,154.005
C08467=1081.659,217.655,422.617,175.154,23.908,154.005
C08468=1081.653,217.406,422.643,175.152,23.905,154.005
C08469=1081.648,217.158,422.668,175.150,23.902,154.004
C08470=1081.642,216.908,422.692,175.147,23.898,154.004
C08471=1081.636,216.661,422.717,175.145,23.895,154.003
C08472=1081.631,216.412,422.743,175.143,23.892,154.003
C08473=1081.625,216.162,422.768,175.141,23.889,154.003
C08474=1081.619,215.914,422.793,175.138,23.885,154.002
C08475=1081.613,215.665,422.817,175.135,23.882,154.002
C08476=1081.608,215.417,422.842,175.133,23.879,154.002
C08477=1081.603,215.167,422.868,175.130,23.876,154.001
C08478=1081.597,214.919,422.893,175.128,23.872,154.001
C08479=1081.591,214.670,422.917,175.126,23.870,154.001
C08480=1081.586,214.422,422.942,175.123,23.866,154.000
C08481=1081.580,214.173,422.967,175.121,23.863,154.000
C08482=1081.575,213.925,422.992,175.119,23.859,153.999
C08483=1081.569,213.675,423.017,175.117,23.856,153.999
C08484=1081.563,213.427,423.042,175.114,23.853,153.999
C08485=1081.557,213.178,423.067,175.112,23.850,153.998
C08486=1081.552,212.930,423.092,175.110,23.847,153.998
C08487=1081.546,212.681,423.116,175.107,23.843,153.997
C08488=1081.540,212.433,423.141,175.104,23.840,153.997
C08489=1081.534,212.184,423.166,175.102,23.837,153.997
C08490=1081.530,211.935,423.191,175.100,23.834,153.996
C08491=1081.524,211.686,423.216,175.097,23.830,153.996
C08492=1081.518,211.437,423.240,175.095,23.827,153.996
C08493=1081.512,211.188,423.265,175.093,23.824,153.995
C08494=1081.507,210.940,423.290,175.091,23.821,153.995
C08495=1081.501,210.691,423.314,175.088,23.817,153.995
C08496=1081.496,210.442,423.339,175.086,23.815,153.994
C08497=1081.489,210.194,423.364,175.084,23.811,153.994
C08498=1081.484,209.945,423.388,175.081,23.808,153.993
C08499=1081.478,209.696,423.413,175.079,23.805,153.993
C08500=1081.469,209.299,423.452,175.075,23.800,153.993
C08501=1081.460,208.903,423.491,175.071,23.795,153.992
C08502=1081.451,208.506,423.530,175.068,23.790,153.991
C08503=1081.442,208.110,423.569,175.063,23.784,153.991
C08504=1081.419,207.078,423.669,174.969,23.734,153.993
C08505=1081.413,206.829,423.692,174.965,23.731,153.993
C08506=1081.407,206.580,423.717,174.963,23.729,153.993
C08507=1081.402,206.331,423.741,174.960,23.727,153.992
C08508=1081.396,206.083,423.765,174.958,23.724,153.992
C08509=1081.391,205.834,423.788,174.956,23.722,153.992
C08510=1081.385,205.585,423.813,174.953,23.720,153.992
C08511=1081.379,205.336,423.837,174.951,23.718,153.992
C08512=1081.373,205.087,423.861,174.949,23.716,153.992
C08513=1081.368,204.838,423.884,174.946,23.713,153.992
C08514=1081.362,204.590,423.908,174.944,23.711,153.991
C08515=1081.357,204.341,423.932,174.941,23.709,153.991
C08516=1081.352,204.091,423.956,174.939,23.707,153.991
C08517=1081.345,203.843,423.980,174.936,23.704,153.991
C08518=1081.340,203.595,424.004,174.933,23.702,153.991
C08519=1081.335,203.345,424.028,174.931,23.700,153.991
C08520=1081.329,203.097,424.051,174.929,23.697,153.991
C08521=1081.324,202.848,424.075,174.926,23.695,153.990
C08522=1081.318,202.600,424.099,174.924,23.693,153.990
C08523=1081.312,202.350,424.123,174.922,23.691,153.990
C08524=1081.307,202.101,424.146,174.919,23.689,153.990
C08525=1081.301,201.853,424.170,174.917,23.686,153.990
C08526=1081.295,201.604,424.193,174.914,23.684,153.990
C08527=1081.289,201.356,424.217,174.912,23.682,153.990
C08528=1081.284,201.106,424.240,174.910,23.680,153.989
C08529=1081.278,200.857,424.265,174.907,23.677,153.989
C08530=1081.273,200.608,424.288,174.905,23.675,153.989
C08531=1081.267,200.360,424.312,174.902,23.673,153.989
C08532=1081.261,200.111,424.335,174.900,23.671,153.989
C08533=1081.256,199.863,424.359,174.898,23.669,153.989
C08534=1081.250,199.614,424.382,174.895,23.667,153.989
C08535=1081.243,199.365,424.406,174.893,23.665,153.988
C08536=1081.238,199.115,424.429,174.890,23.662,153.988
C08537=1081.232,198.867,424.453,174.888,23.660,153.988
C08538=1081.227,198.618,424.477,174.885,23.658,153.988
C08539=1081.222,198.369,424.500,174.882,23.655,153.988
C08540=1081.216,198.121,424.523,174.880,23.653,153.988
C08541=1081.211,197.872,424.547,174.878,23.651,153.988
C08542=1081.205,197.623,424.570,174.875,23.649,153.987
C08543=1081.199,197.374,424.593,174.873,23.646,153.987
C08544=1081.194,197.125,424.617,174.871,23.644,153.987
C08545=1081.188,196.877,424.641,174.868,23.642,153.987
C08546=1081.181,196.627,424.664,174.866,23.640,153.987
C08547=1081.176,196.378,424.687,174.863,23.638,153.987
C08548=1081.171,196.129,424.710,174.861,23.635,153.987
C08549=1081.165,195.881,424.734,174.859,23.633,153.986
C08550=1081.159,195.632,424.757,174.856,23.631,153.986
C08551=1081.154,195.383,424.781,174.854,23.629,153.986
C08552=1081.148,195.135,424.804,174.851,23.627,153.986
C08553=1081.142,194.886,424.827,174.849,23.625,153.986
C08554=1081.137,194.636,424.851,174.847,23.623,153.986
C08555=1081.131,194.388,424.874,174.844,23.620,153.986
C08556=1081.126,194.139,424.897,174.842,23.618,153.986
C08557=1081.120,193.890,424.920,174.840,23.616,153.985
C08558=1081.115,193.641,424.944,174.837,23.614,153.985
C08559=1081.109,193.392,424.967,174.835,23.611,153.985
C08560=1081.103,193.143,424.990,174.832,23.609,153.985
C08561=1081.098,192.894,425.013,174.830,23.607,153.985
C08562=1081.093,192.645,425.036,174.828,23.605,153.985
C08563=1081.087,192.397,425.060,174.826,23.603,153.985
C08564=1081.081,192.148,425.083,174.824,23.601,153.984
C08565=1081.075,191.869,425.109,174.821,23.598,153.984
C08566=1081.068,191.589,425.134,174.818,23.595,153.984
C08567=1081.063,191.310,425.161,174.816,23.593,153.984
C08568=1081.057,191.030,425.186,174.813,23.590,153.984
C08569=1081.051,190.781,425.209,174.810,23.588,153.984
C08570=1081.045,190.532,425.232,174.808,23.586,153.983
C08571=1081.040,190.283,425.255,174.806,23.583,153.983
C08572=1081.034,190.035,425.280,174.803,23.581,153.983
C08573=1081.029,189.786,425.302,174.801,23.579,153.983
C08574=1081.023,189.537,425.325,174.799,23.577,153.983
C08575=1081.018,189.289,425.348,174.797,23.575,153.983
C08576=1081.012,189.040,425.371,174.795,23.573,153.982
C08577=1081.007,188.791,425.394,174.792,23.570,153.982
C08578=1081.002,188.541,425.417,174.790,23.568,153.982
C08579=1080.996,188.292,425.440,174.788,23.566,153.982
C08580=1080.990,188.043,425.463,174.785,23.564,153.982
C08581=1080.985,187.795,425.486,174.783,23.561,153.982
C08582=1080.979,187.546,425.508,174.781,23.559,153.982
C08583=1080.974,187.297,425.532,174.778,23.557,153.981
C08584=1080.969,187.048,425.555,174.776,23.555,153.981
C08585=1080.963,186.799,425.578,174.773,23.552,153.981
C08586=1080.957,186.550,425.600,174.771,23.550,153.981
C08587=1080.951,186.302,425.623,174.769,23.548,153.981
C08588=1080.946,186.053,425.646,174.767,23.545,153.981
C08589=1080.942,185.804,425.669,174.764,23.543,153.980
C08590=1080.936,185.555,425.692,174.763,23.541,153.980
C08591=1080.930,185.306,425.715,174.760,23.539,153.980
C08592=1080.924,185.057,425.738,174.758,23.537,153.980
C08593=1080.919,184.809,425.760,174.756,23.535,153.980
C08594=1080.914,184.559,425.782,174.753,23.532,153.980
C08595=1080.907,184.311,425.805,174.751,23.530,153.980
C08596=1080.902,184.062,425.828,174.748,23.528,153.980
C08597=1080.896,183.813,425.851,174.746,23.526,153.979
C08598=1080.890,183.564,425.874,174.744,23.524,153.979
C08599=1080.885,183.314,425.896,174.741,23.522,153.979
C08600=1080.878,183.066,425.918,174.739,23.519,153.979
C08601=1080.873,182.817,425.941,174.737,23.518,153.979
C08602=1080.868,182.568,425.963,174.735,23.515,153.979
C08603=1080.862,182.319,425.986,174.732,23.514,153.979
C08604=1080.856,182.071,426.008,174.730,23.511,153.979
C08605=1080.850,181.821,426.031,174.728,23.509,153.978
C08606=1080.844,181.572,426.054,174.725,23.507,153.978
C08607=1080.839,181.323,426.076,174.723,23.505,153.978
C08608=1080.833,181.074,426.098,174.721,23.502,153.978
C08609=1080.827,180.826,426.121,174.718,23.500,153.978
C08610=1080.822,180.577,426.144,174.717,23.498,153.978
C08611=1080.816,180.327,426.166,174.714,23.496,153.978
C08612=1080.810,180.079,426.188,174.712,23.494,153.977
C08613=1080.804,179.829,426.210,174.710,23.492,153.977
C08614=1080.799,179.581,426.233,174.707,23.490,153.977
C08615=1080.793,179.333,426.255,174.705,23.488,153.977
C08616=1080.787,179.083,426.278,174.702,23.486,153.977
C08617=1080.782,178.834,426.301,174.700,23.483,153.977
C08618=1080.775,178.585,426.322,174.699,23.481,153.977
C08619=1080.770,178.337,426.345,174.696,23.479,153.976
C08620=1080.765,178.087,426.367,174.694,23.477,153.976
C08621=1080.759,177.838,426.390,174.692,23.475,153.976
C08622=1080.753,177.589,426.412,174.689,23.473,153.976
C08623=1080.748,177.341,426.434,174.687,23.470,153.976
C08624=1080.742,177.091,426.456,174.684,23.468,153.976
C08625=1080.736,176.843,426.479,174.683,23.466,153.976
C08626=1080.731,176.593,426.501,174.681,23.464,153.975
C08627=1080.725,176.345,426.524,174.678,23.462,153.975
C08628=1080.719,176.096,426.545,174.676,23.460,153.975
C08629=1080.713,175.816,426.570,174.674,23.457,153.975
C08630=1080.707,175.537,426.595,174.671,23.455,153.975
C08631=1080.701,175.257,426.620,174.668,23.452,153.975
C08632=1080.694,174.977,426.645,174.666,23.450,153.975
C08633=1080.689,174.728,426.667,174.663,23.448,153.975
C08634=1080.683,174.479,426.690,174.662,23.446,153.974
C08635=1080.677,174.230,426.711,174.659,23.444,153.974
C08636=1080.672,173.981,426.734,174.657,23.442,153.974
C08637=1080.665,173.732,426.756,174.655,23.439,153.974
C08638=1080.661,173.483,426.778,174.652,23.437,153.974
C08639=1080.655,173.234,426.800,174.650,23.435,153.974
C08640=1080.649,172.985,426.822,174.649,23.433,153.973
C08641=1080.644,172.736,426.844,174.646,23.430,153.973
C08642=1080.638,172.487,426.866,174.644,23.428,153.973
C08643=1080.632,172.238,426.889,174.642,23.426,153.973
C08644=1080.627,171.989,426.911,174.639,23.424,153.973
C08645=1080.621,171.740,426.932,174.638,23.422,153.973
C08646=1080.616,171.491,426.954,174.635,23.420,153.972
C08647=1080.610,171.242,426.976,174.633,23.417,153.972
C08648=1080.604,170.993,426.999,174.631,23.415,153.972
C08649=1080.600,170.744,427.021,174.628,23.413,153.972
C08650=1080.593,170.495,427.042,174.627,23.411,153.972
C08651=1080.589,170.246,427.064,174.624,23.409,153.972
C08652=1080.582,169.997,427.086,174.622,23.406,153.972
C08653=1080.577,169.748,427.109,174.620,23.404,153.971
C08654=1080.571,169.500,427.130,174.617,23.402,153.971
C08655=1080.566,169.250,427.152,174.616,23.400,153.971
C08656=1080.561,169.001,427.174,174.614,23.398,153.971
C08657=1080.555,168.752,427.196,174.611,23.396,153.971
C08658=1080.550,168.503,427.218,174.609,23.393,153.971
C08659=1080.544,168.254,427.239,174.607,23.391,153.970
C08660=1080.539,168.006,427.262,174.605,23.389,153.970
C08661=1080.532,167.757,427.283,174.603,23.387,153.970
C08662=1080.528,167.508,427.305,174.600,23.384,153.970
C08663=1080.521,167.259,427.327,174.598,23.382,153.970
C08664=1080.517,167.010,427.349,174.596,23.380,153.970
C08665=1080.510,166.761,427.370,174.594,23.378,153.970
C08666=1080.506,166.512,427.392,174.592,23.376,153.969
C08667=1080.499,166.263,427.414,174.590,23.373,153.969
C08668=1080.495,166.014,427.436,174.587,23.371,153.969
C08669=1080.488,165.765,427.457,174.586,23.369,153.969
C08670=1080.484,165.516,427.479,174.584,23.367,153.969
C08671=1080.477,165.267,427.501,174.581,23.364,153.969
C08672=1080.473,165.018,427.523,174.579,23.362,153.968
C08673=1080.466,164.769,427.544,174.576,23.360,153.968
C08674=1080.462,164.520,427.566,174.575,23.358,153.968
C08675=1080.455,164.271,427.588,174.573,23.355,153.968
C08676=1080.451,164.022,427.610,174.570,23.353,153.968
C08677=1080.445,163.773,427.631,174.568,23.351,153.968
C08678=1080.440,163.524,427.653,174.567,23.349,153.967
C08679=1080.434,163.275,427.674,174.564,23.347,153.967
C08680=1080.429,163.025,427.696,174.562,23.344,153.967
C08681=1080.423,162.777,427.717,174.560,23.342,153.967
C08682=1080.419,162.528,427.739,174.558,23.340,153.967
C08683=1080.412,162.279,427.761,174.556,23.338,153.966
C08684=1080.408,162.030,427.783,174.554,23.335,153.966
C08685=1080.401,161.781,427.804,174.551,23.333,153.966
C08686=1080.396,161.532,427.825,174.550,23.331,153.966
C08687=1080.391,161.282,427.847,174.548,23.329,153.966
C08688=1080.385,161.034,427.868,174.545,23.326,153.966
C08689=1080.380,160.785,427.890,174.543,23.324,153.965
C08690=1080.373,160.536,427.911,174.541,23.322,153.965
C08691=1080.368,160.287,427.932,174.539,23.320,153.965
C08692=1080.363,160.037,427.954,174.537,23.318,153.965
C08693=1080.356,159.757,427.979,174.534,23.315,153.965
C08694=1080.350,159.477,428.002,174.532,23.313,153.965
C08695=1080.344,159.197,428.026,174.530,23.310,153.964
C08696=1080.337,158.917,428.050,174.527,23.308,153.964
C08697=1080.332,158.668,428.071,174.525,23.305,153.964
C08698=1080.326,158.419,428.093,174.524,23.304,153.964
C08699=1080.320,158.170,428.114,174.521,23.301,153.964
C08700=1080.314,157.920,428.135,174.519,23.299,153.964
C08701=1080.309,157.672,428.156,174.517,23.297,153.963
C08702=1080.304,157.423,428.178,174.515,23.295,153.963
C08703=1080.298,157.173,428.199,174.513,23.293,153.963
C08704=1080.292,156.925,428.220,174.511,23.290,153.963
C08705=1080.287,156.676,428.241,174.509,23.289,153.963
C08706=1080.281,156.426,428.262,174.507,23.286,153.963
C08707=1080.275,156.178,428.284,174.505,23.284,153.962
C08708=1080.269,155.929,428.305,174.502,23.281,153.962
C08709=1080.264,155.680,428.326,174.501,23.280,153.962
C08710=1080.259,155.431,428.348,174.498,23.277,153.962
C08711=1080.253,155.181,428.369,174.496,23.275,153.962
C08712=1080.248,154.932,428.390,174.495,23.273,153.962
C08713=1080.243,154.683,428.410,174.492,23.271,153.962
C08714=1080.236,154.434,428.432,174.490,23.269,153.961
C08715=1080.231,154.185,428.453,174.489,23.267,153.961
C08716=1080.225,153.936,428.474,174.486,23.265,153.961
C08717=1080.219,153.687,428.496,174.484,23.262,153.961
C08718=1080.214,153.438,428.516,174.482,23.260,153.961
C08719=1080.208,153.189,428.538,174.480,23.258,153.961
C08720=1080.203,152.940,428.558,174.478,23.255,153.960
C08721=1080.197,152.691,428.580,174.475,23.253,153.960
C08722=1080.191,152.441,428.600,174.474,23.251,153.960
C08723=1080.186,152.192,428.621,174.472,23.249,153.960
C08724=1080.181,151.944,428.642,174.469,23.247,153.960
C08725=1080.175,151.695,428.662,174.468,23.244,153.960
C08726=1080.168,151.446,428.684,174.466,23.242,153.959
C08727=1080.163,151.197,428.704,174.463,23.240,153.959
C08728=1080.158,150.948,428.726,174.462,23.238,153.959
C08729=1080.152,150.698,428.747,174.460,23.236,153.959
C08730=1080.146,150.449,428.767,174.457,23.234,153.959
C08731=1080.141,150.201,428.788,174.456,23.232,153.959
C08732=1080.136,149.952,428.809,174.454,23.229,153.958
C08733=1080.130,149.702,428.830,174.451,23.227,153.958
C08734=1080.124,149.453,428.851,174.450,23.225,153.958
C08735=1080.119,149.204,428.872,174.447,23.223,153.958
C08736=1080.113,148.954,428.893,174.445,23.220,153.958
C08737=1080.107,148.706,428.913,174.444,23.218,153.958
C08738=1080.102,148.457,428.934,174.441,23.216,153.957
C08739=1080.096,148.208,428.954,174.439,23.213,153.957
C08740=1080.090,147.959,428.976,174.438,23.212,153.957
C08741=1080.085,147.710,428.997,174.435,23.209,153.957
C08742=1080.080,147.460,429.017,174.433,23.207,153.957
C08743=1080.073,147.212,429.038,174.432,23.205,153.957
C08744=1080.067,146.962,429.059,174.429,23.203,153.956
C08745=1080.062,146.713,429.079,174.427,23.200,153.956
C08746=1080.057,146.464,429.100,174.426,23.198,153.956
C08747=1080.051,146.215,429.120,174.423,23.196,153.956
C08748=1080.045,145.966,429.141,174.421,23.194,153.956
C08749=1080.040,145.717,429.162,174.419,23.192,153.956
C08750=1080.034,145.468,429.183,174.417,23.190,153.955
C08751=1080.028,145.219,429.203,174.416,23.188,153.955
C08752=1080.022,144.969,429.223,174.413,23.185,153.955
C08753=1080.017,144.721,429.245,174.411,23.183,153.955
C08754=1080.012,144.472,429.265,174.410,23.181,153.955
C08755=1080.006,144.223,429.285,174.407,23.179,153.955
C08756=1080.000,143.974,429.306,174.405,23.176,153.954
C08757=1079.994,143.693,429.330,174.403,23.174,153.954
C08758=1079.987,143.413,429.352,174.400,23.171,153.954
C08759=1079.981,143.132,429.376,174.398,23.169,153.954
C08760=1079.974,142.852,429.398,174.397,23.167,153.954
C08761=1079.969,142.603,429.419,174.394,23.165,153.953
C08762=1079.964,142.353,429.439,174.392,23.162,153.953
C08763=1079.958,142.105,429.459,174.391,23.160,153.953
C08764=1079.953,141.856,429.480,174.389,23.158,153.953
C08765=1079.946,141.606,429.501,174.386,23.155,153.953
C08766=1079.941,141.357,429.522,174.385,23.153,153.952
C08767=1079.935,141.108,429.542,174.383,23.151,153.952
C08768=1079.930,140.859,429.562,174.381,23.149,153.952
C08769=1079.925,140.610,429.583,174.379,23.147,153.952
C08770=1079.919,140.361,429.603,174.377,23.144,153.952
C08771=1079.913,140.112,429.624,174.375,23.142,153.952
C08772=1079.907,139.863,429.644,174.373,23.140,153.951
C08773=1079.902,139.614,429.664,174.370,23.137,153.951
C08774=1079.896,139.365,429.684,174.369,23.136,153.951
C08775=1079.891,139.115,429.704,174.367,23.133,153.951
C08776=1079.885,138.866,429.725,174.365,23.131,153.951
C08777=1079.879,138.617,429.745,174.363,23.129,153.951
C08778=1079.874,138.368,429.765,174.361,23.126,153.950
C08779=1079.868,138.119,429.785,174.359,23.125,153.950
C08780=1079.862,137.869,429.806,174.357,23.122,153.950
C08781=1079.856,137.620,429.826,174.356,23.120,153.950
C08782=1079.851,137.371,429.847,174.353,23.118,153.950
C08783=1079.845,137.123,429.867,174.351,23.115,153.949
C08784=1079.840,136.873,429.887,174.350,23.113,153.949
C08785=1079.834,136.624,429.906,174.347,23.111,153.949
C08786=1079.829,136.375,429.927,174.346,23.109,153.949
C08787=1079.823,136.126,429.947,174.344,23.107,153.949
C08788=1079.818,135.877,429.967,174.342,23.104,153.948
C08789=1079.812,135.628,429.987,174.340,23.102,153.948
C08790=1079.806,135.379,430.007,174.338,23.100,153.948
C08791=1079.800,135.129,430.028,174.336,23.098,153.948
C08792=1079.794,134.880,430.048,174.334,23.095,153.948
C08793=1079.789,134.631,430.068,174.333,23.093,153.948
C08794=1079.783,134.382,430.088,174.330,23.091,153.947
C08795=1079.778,134.132,430.108,174.328,23.089,153.947
C08796=1079.772,133.884,430.128,174.327,23.086,153.947
C08797=1079.767,133.634,430.148,174.324,23.084,153.947
C08798=1079.761,133.386,430.168,174.323,23.082,153.947
C08799=1079.755,133.136,430.188,174.321,23.079,153.946
C08800=1079.750,132.887,430.208,174.319,23.077,153.946
C08801=1079.744,132.638,430.228,174.317,23.075,153.946
C08802=1079.738,132.389,430.249,174.315,23.073,153.946
C08803=1079.733,132.140,430.268,174.313,23.071,153.946
C08804=1079.727,131.891,430.288,174.311,23.068,153.946
C08805=1079.721,131.642,430.308,174.310,23.066,153.945
C08806=1079.716,131.392,430.328,174.307,23.064,153.945
C08807=1079.710,131.144,430.348,174.306,23.062,153.945
C08808=1079.704,130.895,430.368,174.304,23.060,153.945
C08809=1079.698,130.645,430.387,174.302,23.058,153.945
C08810=1079.693,130.396,430.407,174.300,23.055,153.945
C08811=1079.687,130.147,430.427,174.297,23.053,153.944
C08812=1079.681,129.898,430.447,174.296,23.051,153.944
C08813=1079.675,129.648,430.467,174.294,23.048,153.944
C08814=1079.669,129.399,430.486,174.292,23.047,153.944
C08815=1079.664,129.150,430.507,174.290,23.044,153.944
C08816=1079.658,128.900,430.526,174.289,23.042,153.943
C08817=1079.652,128.652,430.546,174.286,23.040,153.943
C08818=1079.646,128.402,430.565,174.285,23.038,153.943
C08819=1079.640,128.153,430.585,174.283,23.036,153.943
C08820=1079.635,127.904,430.605,174.281,23.033,153.943
C08821=1079.629,127.624,430.627,174.279,23.031,153.942
C08822=1079.623,127.343,430.649,174.277,23.028,153.942
C08823=1079.616,127.063,430.672,174.275,23.026,153.942
C08824=1079.610,126.782,430.694,174.272,23.023,153.942
C08825=1079.604,126.533,430.713,174.270,23.021,153.942
C08826=1079.598,126.284,430.733,174.269,23.019,153.941
C08827=1079.592,126.035,430.752,174.267,23.016,153.941
C08828=1079.586,125.786,430.772,174.265,23.014,153.941
C08829=1079.581,125.536,430.792,174.263,23.012,153.941
C08830=1079.575,125.288,430.812,174.261,23.010,153.941
C08831=1079.569,125.038,430.831,174.259,23.007,153.940
C08832=1079.564,124.788,430.851,174.258,23.005,153.940
C08833=1079.558,124.540,430.871,174.256,23.003,153.940
C08834=1079.552,124.290,430.890,174.254,23.001,153.940
C08835=1079.547,124.042,430.909,174.252,22.998,153.940
C08836=1079.541,123.793,430.929,174.251,22.996,153.939
C08837=1079.536,123.543,430.948,174.248,22.994,153.939
C08838=1079.530,123.294,430.968,174.247,22.992,153.939
C08839=1079.524,123.045,430.987,174.245,22.989,153.939
C08840=1079.519,122.795,431.007,174.243,22.987,153.939
C08841=1079.513,122.546,431.027,174.241,22.984,153.938
C08842=1079.507,122.297,431.046,174.240,22.983,153.938
C08843=1079.502,122.048,431.065,174.237,22.980,153.938
C08844=1079.496,121.799,431.085,174.235,22.978,153.938
C08845=1079.491,121.550,431.104,174.234,22.976,153.938
C08846=1079.485,121.301,431.123,174.231,22.973,153.938
C08847=1079.479,121.051,431.143,174.230,22.971,153.937
C08848=1079.473,120.802,431.163,174.228,22.969,153.937
C08849=1079.467,120.553,431.182,174.226,22.966,153.937
C08850=1079.462,120.303,431.201,174.224,22.964,153.937
C08851=1079.457,120.055,431.220,174.223,22.962,153.936
C08852=1079.451,119.806,431.240,174.221,22.959,153.936
C08853=1079.446,119.556,431.260,174.219,22.958,153.936
C08854=1079.440,119.307,431.279,174.217,22.955,153.936
C08855=1079.434,119.057,431.298,174.215,22.953,153.936
C08856=1079.429,118.809,431.318,174.213,22.950,153.935
C08857=1079.423,118.560,431.337,174.212,22.948,153.935
C08858=1079.418,118.310,431.356,174.210,22.945,153.935
C08859=1079.412,118.061,431.376,174.208,22.943,153.935
C08860=1079.406,117.811,431.395,174.206,22.941,153.935
C08861=1079.401,117.563,431.414,174.205,22.939,153.934
C08862=1079.395,117.314,431.434,174.202,22.937,153.934
C08863=1079.389,117.065,431.453,174.201,22.934,153.934
C08864=1079.384,116.815,431.472,174.199,22.932,153.934
C08865=1079.379,116.566,431.491,174.198,22.929,153.933
C08866=1079.373,116.317,431.510,174.195,22.927,153.933
C08867=1079.367,116.067,431.530,174.194,22.925,153.933
C08868=1079.362,115.818,431.549,174.193,22.923,153.933
C08869=1079.357,115.569,431.568,174.190,22.920,153.933
C08870=1079.351,115.320,431.587,174.189,22.918,153.932
C08871=1079.345,115.070,431.606,174.187,22.915,153.932
C08872=1079.339,114.821,431.625,174.185,22.914,153.932
C08873=1079.334,114.572,431.644,174.183,22.911,153.932
C08874=1079.329,114.323,431.664,174.182,22.909,153.932
C08875=1079.323,114.073,431.683,174.180,22.906,153.931
C08876=1079.317,113.825,431.703,174.178,22.904,153.931
C08877=1079.311,113.576,431.721,174.176,22.901,153.931
C08878=1079.305,113.327,431.740,174.175,22.900,153.931
C08879=1079.300,113.077,431.759,174.172,22.897,153.930
C08880=1079.294,112.827,431.778,174.171,22.895,153.930
C08881=1079.289,112.579,431.797,174.169,22.892,153.930
C08882=1079.283,112.329,431.816,174.167,22.890,153.930
C08883=1079.277,112.080,431.835,174.165,22.888,153.930
C08884=1079.272,111.831,431.854,174.164,22.885,153.929
C08885=1079.266,111.550,431.875,174.162,22.883,153.929
C08886=1079.259,111.270,431.897,174.159,22.880,153.929
C08887=1079.252,110.989,431.918,174.158,22.878,153.929
C08888=1079.246,110.709,431.939,174.156,22.875,153.928
C08889=1079.240,110.459,431.959,174.154,22.873,153.928
C08890=1079.234,110.211,431.977,174.152,22.871,153.928
C08891=1079.229,109.962,431.996,174.150,22.868,153.928
C08892=1079.223,109.712,432.015,174.149,22.866,153.928
C08893=1079.217,109.462,432.033,174.147,22.864,153.927
C08894=1079.212,109.214,432.052,174.145,22.862,153.927
C08895=1079.206,108.964,432.071,174.144,22.859,153.927
C08896=1079.200,108.715,432.090,174.142,22.857,153.927
C08897=1079.195,108.466,432.109,174.140,22.855,153.927
C08898=1079.189,108.217,432.128,174.138,22.852,153.926
C08899=1079.183,107.967,432.146,174.137,22.850,153.926
C08900=1079.178,107.718,432.165,174.134,22.848,153.926
C08901=1079.172,107.469,432.184,174.133,22.845,153.926
C08902=1079.166,107.220,432.203,174.131,22.843,153.926
C08903=1079.161,106.971,432.221,174.130,22.841,153.925
C08904=1079.154,106.721,432.240,174.128,22.839,153.925
C08905=1079.149,106.472,432.259,174.126,22.836,153.925
C08906=1079.144,106.223,432.278,174.125,22.834,153.925
C08907=1079.138,105.973,432.296,174.122,22.831,153.924
C08908=1079.132,105.724,432.315,174.121,22.829,153.924
C08909=1079.127,105.475,432.334,174.119,22.826,153.924
C08910=1079.120,105.226,432.353,174.117,22.825,153.924
C08911=1079.115,104.976,432.371,174.115,22.822,153.924
C08912=1079.109,104.728,432.389,174.114,22.820,153.923
C08913=1079.103,104.478,432.409,174.113,22.817,153.923
C08914=1079.098,104.228,432.427,174.110,22.815,153.923
C08915=1079.092,103.980,432.445,174.109,22.813,153.923
C08916=1079.087,103.730,432.465,174.107,22.810,153.923
C08917=1079.081,103.481,432.482,174.105,22.808,153.922
C08918=1079.075,103.232,432.501,174.103,22.805,153.922
C08919=1079.069,102.983,432.520,174.102,22.803,153.922
C08920=1079.064,102.733,432.538,174.100,22.801,153.922
C08921=1079.058,102.484,432.557,174.098,22.799,153.921
C08922=1079.053,102.235,432.575,174.097,22.796,153.921
C08923=1079.047,101.986,432.594,174.095,22.794,153.921
C08924=1079.041,101.737,432.613,174.093,22.792,153.921
C08925=1079.036,101.487,432.631,174.091,22.789,153.920
C08926=1079.030,101.238,432.650,174.090,22.787,153.920
C08927=1079.025,100.989,432.668,174.089,22.784,153.920
C08928=1079.018,100.739,432.687,174.086,22.782,153.920
C08929=1079.014,100.490,432.705,174.085,22.780,153.919
C08930=1079.007,100.241,432.723,174.083,22.777,153.919
C08931=1079.001,99.991,432.741,174.082,22.775,153.919
C08932=1078.996,99.743,432.760,174.079,22.773,153.919
C08933=1078.990,99.493,432.778,174.078,22.770,153.919
C08934=1078.985,99.244,432.797,174.077,22.769,153.918
C08935=1078.979,98.994,432.815,174.074,22.766,153.918
C08936=1078.973,98.746,432.833,174.073,22.764,153.918
C08937=1078.967,98.496,432.852,174.071,22.761,153.918
C08938=1078.961,98.247,432.870,174.069,22.759,153.918
C08939=1078.956,97.998,432.888,174.068,22.757,153.917
C08940=1078.950,97.748,432.907,174.066,22.754,153.917
C08941=1078.944,97.499,432.925,174.065,22.752,153.917
C08942=1078.938,97.250,432.943,174.062,22.749,153.917
C08943=1078.933,97.001,432.962,174.061,22.747,153.916
C08944=1078.927,96.751,432.979,174.059,22.744,153.916
C08945=1078.921,96.503,432.998,174.058,22.743,153.916
C08946=1078.916,96.253,433.016,174.056,22.740,153.916
C08947=1078.910,96.004,433.035,174.054,22.737,153.915
C08948=1078.904,95.754,433.053,174.053,22.735,153.915
C08949=1078.897,95.474,433.073,174.051,22.733,153.915
C08950=1078.891,95.193,433.093,174.048,22.730,153.915
C08951=1078.885,94.913,433.114,174.047,22.727,153.914
C08952=1078.878,94.632,433.134,174.045,22.725,153.914
C08953=1078.873,94.383,433.153,174.044,22.723,153.914
C08954=1078.867,94.134,433.171,174.042,22.720,153.914
C08955=1078.862,93.885,433.188,174.040,22.717,153.913
C08956=1078.856,93.635,433.208,174.038,22.715,153.913
C08957=1078.850,93.386,433.225,174.037,22.713,153.913
C08958=1078.844,93.136,433.243,174.035,22.710,153.913
C08959=1078.839,92.888,433.262,174.033,22.708,153.913
C08960=1078.833,92.638,433.280,174.032,22.706,153.912
C08961=1078.828,92.389,433.298,174.030,22.704,153.912
C08962=1078.822,92.140,433.315,174.028,22.701,153.912
C08963=1078.816,91.890,433.334,174.027,22.699,153.912
C08964=1078.811,91.641,433.352,174.025,22.696,153.911
C08965=1078.805,91.392,433.370,174.024,22.694,153.911
C08966=1078.800,91.142,433.388,174.022,22.691,153.911
C08967=1078.794,90.892,433.406,174.020,22.689,153.911
C08968=1078.788,90.644,433.424,174.019,22.687,153.910
C08969=1078.782,90.394,433.442,174.017,22.684,153.910
C08970=1078.776,90.145,433.460,174.015,22.682,153.910
C08971=1078.770,89.896,433.478,174.014,22.680,153.910
C08972=1078.765,89.647,433.495,174.012,22.677,153.910
C08973=1078.759,89.397,433.513,174.010,22.675,153.909
C08974=1078.753,89.148,433.531,174.009,22.673,153.909
C08975=1078.747,88.899,433.549,174.007,22.670,153.909
C08976=1078.742,88.649,433.568,174.006,22.668,153.909
C08977=1078.736,88.400,433.585,174.003,22.665,153.908
C08978=1078.730,88.150,433.603,174.002,22.663,153.908
C08979=1078.725,87.901,433.621,174.001,22.661,153.908
C08980=1078.719,87.652,433.639,173.999,22.658,153.908
C08981=1078.713,87.403,433.656,173.997,22.656,153.907
C08982=1078.708,87.154,433.674,173.996,22.654,153.907
C08983=1078.701,86.904,433.692,173.994,22.651,153.907
C08984=1078.696,86.655,433.710,173.993,22.649,153.907
C08985=1078.689,86.406,433.728,173.990,22.646,153.907
C08986=1078.684,86.157,433.745,173.989,22.644,153.906
C08987=1078.678,85.908,433.763,173.988,22.642,153.906
C08988=1078.672,85.658,433.781,173.985,22.639,153.906
C08989=1078.667,85.409,433.799,173.984,22.637,153.906
C08990=1078.661,85.159,433.816,173.983,22.635,153.905
C08991=1078.655,84.910,433.834,173.981,22.632,153.905
C08992=1078.650,84.661,433.852,173.979,22.630,153.905
C08993=1078.643,84.411,433.870,173.977,22.627,153.905
C08994=1078.638,84.162,433.887,173.976,22.625,153.904
C08995=1078.632,83.913,433.905,173.975,22.623,153.904
C08996=1078.626,83.663,433.923,173.972,22.620,153.904
C08997=1078.621,83.414,433.940,173.971,22.618,153.904
C08998=1078.615,83.165,433.958,173.970,22.615,153.903
C08999=1078.609,82.915,433.975,173.968,22.613,153.903
C09000=1078.604,82.666,433.992,173.966,22.611,153.903
C09001=1078.598,82.417,434.010,173.965,22.608,153.903
C09002=1078.592,82.167,434.028,173.963,22.605,153.902
C09003=1078.587,81.918,434.046,173.962,22.604,153.902
C09004=1078.581,81.669,434.063,173.960,22.601,153.902
C09005=1078.575,81.419,434.081,173.958,22.598,153.902
C09006=1078.570,81.170,434.099,173.957,22.596,153.901
C09007=1078.564,80.921,434.116,173.955,22.594,153.901
C09008=1078.559,80.672,434.133,173.953,22.591,153.901
C09009=1078.553,80.422,434.151,173.952,22.589,153.901
C09010=1078.547,80.173,434.169,173.950,22.586,153.900
C09011=1078.542,79.924,434.186,173.949,22.584,153.900
C09012=1078.536,79.674,434.204,173.947,22.582,153.900
C09013=1078.529,79.394,434.223,173.945,22.579,153.900
C09014=1078.523,79.113,434.243,173.943,22.576,153.899
C09015=1078.517,78.833,434.262,173.942,22.574,153.899
C09016=1078.510,78.553,434.282,173.940,22.571,153.899
C09017=1078.505,78.304,434.300,173.939,22.568,153.899
C09018=1078.499,78.054,434.318,173.936,22.565,153.898
C09019=1078.493,77.804,434.334,173.935,22.564,153.898
C09020=1078.487,77.555,434.352,173.934,22.561,153.898
C09021=1078.481,77.306,434.370,173.932,22.558,153.898
C09022=1078.476,77.057,434.387,173.930,22.556,153.897
C09023=1078.470,76.807,434.403,173.929,22.554,153.897
C09024=1078.464,76.558,434.421,173.927,22.551,153.897
C09025=1078.458,76.308,434.439,173.926,22.549,153.897
C09026=1078.453,76.059,434.456,173.924,22.547,153.896
C09027=1078.447,75.810,434.473,173.922,22.544,153.896
C09028=1078.441,75.561,434.490,173.921,22.542,153.896
C09029=1078.435,75.311,434.507,173.920,22.540,153.896
C09030=1078.430,75.062,434.525,173.917,22.537,153.895
C09031=1078.424,74.813,434.542,173.916,22.534,153.895
C09032=1078.418,74.563,434.559,173.915,22.532,153.895
C09033=1078.412,74.314,434.577,173.913,22.530,153.895
C09034=1078.407,74.065,434.594,173.911,22.527,153.894
C09035=1078.401,73.815,434.611,173.910,22.525,153.894
C09036=1078.395,73.566,434.628,173.908,22.522,153.894
C09037=1078.389,73.316,434.646,173.907,22.520,153.894
C09038=1078.384,73.067,434.663,173.905,22.518,153.893
C09039=1078.378,72.818,434.680,173.903,22.515,153.893
C09040=1078.372,72.568,434.697,173.902,22.513,153.893
C09041=1078.367,72.319,434.714,173.901,22.510,153.893
C09042=1078.360,72.069,434.731,173.899,22.508,153.892
C09043=1078.355,71.820,434.749,173.897,22.506,153.892
C09044=1078.349,71.571,434.766,173.896,22.503,153.892
C09045=1078.343,71.322,434.782,173.895,22.501,153.892
C09046=1078.338,71.073,434.800,173.893,22.498,153.891
C09047=1078.333,70.823,434.817,173.891,22.496,153.891
C09048=1078.326,70.574,434.834,173.890,22.494,153.891
C09049=1078.321,70.324,434.851,173.888,22.491,153.891
C09050=1078.315,70.075,434.869,173.887,22.488,153.890
C09051=1078.309,69.826,434.885,173.885,22.486,153.890
C09052=1078.304,69.577,434.902,173.883,22.484,153.890
C09053=1078.298,69.327,434.919,173.882,22.481,153.890
C09054=1078.291,69.077,434.937,173.881,22.479,153.889
C09055=1078.286,68.828,434.953,173.878,22.477,153.889
C09056=1078.280,68.579,434.970,173.877,22.474,153.889
C09057=1078.275,68.329,434.987,173.876,22.472,153.889
C09058=1078.269,68.080,435.003,173.874,22.469,153.888
C09059=1078.263,67.831,435.021,173.872,22.467,153.888
C09060=1078.257,67.581,435.038,173.871,22.465,153.888
C09061=1078.251,67.332,435.055,173.869,22.462,153.888
C09062=1078.245,67.083,435.071,173.868,22.459,153.887
C09063=1078.240,66.833,435.088,173.866,22.457,153.887
C09064=1078.234,66.584,435.105,173.865,22.455,153.887
C09065=1078.229,66.335,435.122,173.863,22.452,153.887
C09066=1078.222,66.086,435.139,173.862,22.450,153.886
C09067=1078.217,65.836,435.156,173.860,22.448,153.886
C09068=1078.211,65.586,435.173,173.858,22.445,153.886
C09069=1078.205,65.337,435.190,173.857,22.442,153.886
C09070=1078.199,65.088,435.206,173.856,22.440,153.885
C09071=1078.194,64.838,435.223,173.854,22.437,153.885
C09072=1078.188,64.589,435.240,173.852,22.435,153.885
C09073=1078.182,64.340,435.257,173.851,22.433,153.884
C09074=1078.177,64.090,435.273,173.849,22.430,153.884
C09075=1078.170,63.842,435.290,173.848,22.428,153.884
C09076=1078.164,63.591,435.308,173.846,22.426,153.884
C09077=1078.158,63.311,435.326,173.844,22.423,153.884
C09078=1078.151,63.031,435.345,173.843,22.420,153.883
C09079=1078.145,62.750,435.363,173.841,22.418,153.883
C09080=1078.138,62.469,435.383,173.840,22.415,153.883
C09081=1078.132,62.220,435.399,173.838,22.412,153.882
C09082=1078.126,61.970,435.416,173.836,22.410,153.882
C09083=1078.121,61.721,435.432,173.835,22.408,153.882
C09084=1078.114,61.472,435.449,173.833,22.405,153.882
C09085=1078.108,61.223,435.465,173.832,22.403,153.881
C09086=1078.103,60.973,435.482,173.830,22.401,153.881
C09087=1078.097,60.724,435.498,173.828,22.398,153.881
C09088=1078.091,60.474,435.515,173.827,22.395,153.881
C09089=1078.085,60.225,435.531,173.826,22.393,153.880
C09090=1078.079,59.976,435.549,173.824,22.391,153.880
C09091=1078.073,59.726,435.565,173.822,22.388,153.880
C09092=1078.067,59.477,435.581,173.821,22.386,153.880
C09093=1078.061,59.228,435.597,173.820,22.383,153.879
C09094=1078.056,58.978,435.614,173.818,22.381,153.879
C09095=1078.050,58.729,435.631,173.816,22.379,153.879
C09096=1078.044,58.480,435.648,173.815,22.376,153.879
C09097=1078.038,58.230,435.664,173.814,22.374,153.878
C09098=1078.033,57.981,435.681,173.812,22.371,153.878
C09099=1078.027,57.731,435.697,173.810,22.369,153.878
C09100=1078.021,57.482,435.713,173.809,22.367,153.878
C09101=1078.015,57.233,435.729,173.807,22.364,153.877
C09102=1078.010,56.983,435.746,173.806,22.362,153.877
C09103=1078.004,56.734,435.763,173.804,22.359,153.877
C09104=1077.998,56.484,435.779,173.803,22.357,153.877
C09105=1077.992,56.235,435.795,173.801,22.354,153.876
